	    IF (#i.ctrl.OFFVAL < #calc.speedmin) AND (#i.ctrl.ITLVAL > #calc.speedmax) THEN
	        #i.ctrl.OFFVAL := #calc.speedmin;
	    END_IF;
	    
	    //Network24: SPEED CONTROL: Determine if initialization routine is required
	    
	    #i.ctrl.init.req := (#i.ctrl.ITLVAL > #calc.speedmin) AND (#i.ctrl.init.dur < 0);
	    
	    //Network25: SPEED CONTROL: Determine the delay SP
	    
	    IF NOT #i.out.run AND #i.ctrl.init.req THEN
	        #i.ctrl.init.delay.in.spon := #i.ctrl.init.dur;
	    END_IF;
	    
	    IF NOT #i.out.run AND NOT #i.ctrl.init.req THEN
	        #i.ctrl.init.delay.in.spon := 0.0;
	    END_IF;
	    
	    IF #i.ctrl.mode OR NOT #ctrl_internal THEN
	        #i.ctrl.init.delay.in.spon := 0.0;
	    END_IF;
	    
	    //Network26: SPEED CONTROL: Delay for holding an init value
	    
	    "AFC_DelayONOFF"(cmd := #i.out.run,
	                     Pulse := #p100ms,
	                     Reset := NOT #i.out.run,
	                     on => #i.ctrl.init.delay.out.on,
	                     Data := #i.ctrl.init.delay);
	    
	    //Network27: SPEED CONTROL: Load output
	    
	    IF NOT #i.ctrl.mode THEN
	        
	        IF NOT #i.out.run THEN
	            
	            IF NOT #ctrl_internal THEN
	                
	                IF #i.ctrl.init.delay.out.on THEN
	                    #i.ctrl.OP := #i.scale.output;
	                END_IF;
	                
	                IF #i.ctrl.init.delay.out.on THEN
	                    #i.ctrl.OP := #i.ctrl.ITLVAL;
	                END_IF;
	                
	            END_IF;
	            
	        ELSIF NOT #ctrl_internal THEN
	            
	             #i.ctrl.OP := #i.ctrl.FUP;
	             
	        ELSE // 20240403: CH - Added "ELSE" for linear control
	             #i.ctrl.OP := #i.scale.output;
	            
	        END_IF;
	        
	    ELSIF #i.ctrl.mode THEN
	        
	         IF NOT #i.out.run AND NOT #i.ctrl.mode THEN
	            #i.ctrl.OP := #i.ctrl.OFFVAL;
	        END_IF;
	        
	    END_IF;
	    
	END_REGION
	
	REGION ARH  NW:28
	    
	    //Network28: ARH: Working hours counter
	    
	    IF #i.status.vfb AND #p1s THEN
	        #i.arh.seconds := #i.arh.seconds + 1;
	    END_IF;
	    
	    #i.arh.hour := #i.arh.seconds >= 3600;
	    
	    IF #i.arh.hour THEN
	        #i.arh.actual := #i.arh.actual + 1;
	        #i.arh.seconds := 0;
	    END_IF;
	    
	    IF #i.arh.resetarh THEN
	        #i.arh.actual := #i.arh.lastmaint := 0;
	    END_IF;
	    
	    #i.arh.difference := #i.arh.actual - #i.arh.lastmaint;
	    
	END_REGION
	
	REGION UNSCALE  NW:29-33
	    
	    //Network29: UNSCALE: Move input
	    
	    #i.unscale.in := #i.ctrl.OP;
	    
	    //Network30: UNSCALE: Cross-check unscaling setup
	    
	    #i.unscale.set := (#i.unscale.inhigh <> #i.unscale.inlow) AND (#i.unscale.outhigh <> #i.unscale.outlow);
	    
	    //Network31: UNSCALE: Determine sign of scaling slope and calculation operands (Hi - Low)
	    
	    IF #i.unscale.set THEN
	        #calc.inspan := #i.unscale.inhigh - #i.unscale.inlow;
	        #calc.outspan := #i.unscale.outhigh - #i.unscale.outlow;
	        #calc.x := #i.unscale.in;
	        IF #calc.inspan > 0 AND #calc.outspan > 0 THEN
	            #calc.sign := TRUE;
	            #calc.ymax := #i.unscale.outhigh;
	            #calc.ymin := #i.unscale.outlow;
	            #calc.xmax := #i.unscale.inhigh;
	            #calc.xmin := #i.unscale.inlow;
	        ELSIF #calc.inspan < 0 AND #calc.outspan < 0 THEN
	            #calc.sign := TRUE;
	            #calc.ymax := #i.unscale.outlow;
	            #calc.ymin := #i.unscale.outhigh;
	            #calc.xmax := #i.unscale.inlow;
	            #calc.xmin := #i.unscale.inhigh;
	        ELSIF #calc.inspan < 0 AND #calc.outspan > 0 THEN
	            #calc.sign := FALSE;
	            #calc.ymax := #i.unscale.outlow;
	            #calc.ymin := #i.unscale.outhigh;
	            #calc.xmax := #i.unscale.inhigh;
	            #calc.xmin := #i.unscale.inlow;
	        ELSE
	            #calc.sign := FALSE;
	            #calc.ymax := #i.unscale.outhigh;
	            #calc.ymin := #i.unscale.outlow;
	            #calc.xmax := #i.unscale.inlow;
	            #calc.xmin := #i.unscale.inhigh;
	        END_IF;
	        #calc.speedmin := #calc.xmin;
	        #calc.speedmax := #calc.xmax;
	    ELSE
	        #calc.inspan := #calc.outspan := #calc.xmax := #calc.xmin
	        := #calc.ymax := #calc.ymin := #calc.speedmin := #calc.speedmax := 0.0;
	    END_IF;
	    
	    //Network32: UNSCALE: Determine output
	    
	    IF #i.unscale.set AND #calc.sign THEN
	        
	        #calc.y := #calc.ymin + ((#calc.ymax - #calc.ymin) * (#calc.x - #calc.xmin) / (#calc.xmax - #calc.xmin));
	        
	        IF #calc.x <= #calc.xmin THEN
	            #calc.y := #calc.ymin;
	        END_IF;
	        
	        IF #calc.x >= #calc.xmax THEN
	            #calc.y := #calc.ymax;
	        END_IF;
	        
	    END_IF;
	    
	    IF #i.unscale.set AND NOT #calc.sign THEN
	        
	        #calc.y := #calc.ymin + ((#calc.ymax - #calc.ymin) * (#calc.xmax - #calc.x) / (#calc.xmax - #calc.xmin));
	        
	        IF #calc.x <= #calc.xmin THEN
	            #calc.y := #calc.ymax;
	        END_IF;
	        
	        IF #calc.x >= #calc.xmax THEN
	            #calc.y := #calc.ymin;
	        END_IF;
	        
	    END_IF;
	    
	    IF #i.unscale.set THEN
	        #i.unscale.output := #calc.y;
	    END_IF;
	    
	    IF NOT #i.unscale.set THEN
	        #i.unscale.output := 0.0;
	    END_IF;
	    
	    //Network33: UNSCALE: Convert to INT
	    
	    #i.out."ref" := REAL_TO_INT(#i.unscale.output);
	    
	END_REGION
	
	REGION UNSCALE  NW:34-35
	    
	    //Network34: ARH: Maintenance required
	    
	    #condSET := #i.arh.difference >= #i.arh.checkafter;
	    #condRESET := (#i.arh.completed AND #i.arh.maintenance) OR NOT #i.arh.enable;
	    
	    #i.arh.maintenance := (#i.arh.maintenance OR #condSET) AND NOT #condRESET;
	    
	    IF #i.arh.completed AND #i.arh.maintenance THEN
	        #i.arh.lastmaint := #i.arh.actual;
	    END_IF;
	    
	    
	    //Network35: STATUS: Maintenance required
	    
	    #i.status.maint := #i.arh.maintenance;
	    
	END_REGION
	
	REGION OUTPUT  NW:36
	    
	    //Network36: Move UDT outputs to FC outputs
	    
	    #run := #i.out.run;
	    #vfb := #i.status.vfb;
	    
	    #reference := #i.out."ref";
	    
	END_REGION
	
	REGION BUTTON  NW:37
	    
	    //Network37: EXTRA: Button treatment
	    
	    IF #i.ind.auto THEN
	        #i.cmd.auto := FALSE;
	    END_IF;
	    
	    IF #i.ind.man THEN
	        #i.cmd.man := FALSE;
	    END_IF;
	    
	    IF #i.ind.start OR #i.ind.auto OR NOT #i.status.ilstart THEN
	        #i.cmd.start := FALSE;
	    END_IF;
	    
	    IF #i.ind.stop OR #i.ind.auto THEN
	        #i.cmd.stop := FALSE;
	    END_IF;
	    
	    IF #i.faults.fpreset THEN
	        #i.faults.fpreset := FALSE;
	    END_IF;
	    
	    IF (#i.arh.seconds = 0) AND (#i.arh.actual = 0) THEN
	        #i.arh.resetarh := FALSE;
	    END_IF;
	    
	END_REGION
END_FUNCTION_BLOCK

FUNCTION_BLOCK "AFB_MotorPID_v3"
{ S7_Optimized_Access := 'TRUE' }
VERSION : 0.1
   VAR_INPUT 
      start { ExternalAccessible := 'False'; ExternalVisible := 'False'; ExternalWritable := 'False'} : Bool;   // "Logic" in order to start
      spsource { ExternalAccessible := 'False'; ExternalVisible := 'False'; ExternalWritable := 'False'} : Bool;   // 0=internal setpoint, 1=external setpoint
      followup { ExternalAccessible := 'False'; ExternalVisible := 'False'; ExternalWritable := 'False'} : Bool;   // 0=motor control from PID, 1=motor setpoint directly from program
      pidrun { ExternalAccessible := 'False'; ExternalVisible := 'False'; ExternalWritable := 'False'} : Bool;   // 0=controller not ready, controller is running
      "fb" { ExternalAccessible := 'False'; ExternalVisible := 'False'; ExternalWritable := 'False'} : Bool;   // Motor's running feedback (1=run, 0=stop)
      mcb { ExternalAccessible := 'False'; ExternalVisible := 'False'; ExternalWritable := 'False'} : Bool;   // Motor circuit breaker (1=ok, 0=fault)
      ctrl { ExternalAccessible := 'False'; ExternalVisible := 'False'; ExternalWritable := 'False'} : Bool;   // Control of motor (1=PLC, 0=Local)
      vfdnotrip { ExternalAccessible := 'False'; ExternalVisible := 'False'; ExternalWritable := 'False'} : Bool;   // VFD health condition (1=ok, 0=fault)
      block { ExternalAccessible := 'False'; ExternalVisible := 'False'; ExternalWritable := 'False'} : Bool;   // Condition that blocks motor operation
      generalackn { ExternalAccessible := 'False'; ExternalVisible := 'False'; ExternalWritable := 'False'} : Bool;   // General acknowledgement
      reset { ExternalAccessible := 'False'; ExternalVisible := 'False'; ExternalWritable := 'False'} : Bool;   // Option that resets the faults
      mute { ExternalAccessible := 'False'; ExternalVisible := 'False'; ExternalWritable := 'False'} : Bool;   // Mute siren
      autoset { ExternalAccessible := 'False'; ExternalVisible := 'False'; ExternalWritable := 'False'} : Bool;   // Option that sets the motor to auto mode (Used for mass auto set)
      manualset { ExternalAccessible := 'False'; ExternalVisible := 'False'; ExternalWritable := 'False'} : Bool;   // Option that sets the motor to manual mode (Used for mass manual set)
      p1s { ExternalAccessible := 'False'; ExternalVisible := 'False'; ExternalWritable := 'False'} : Bool;   // Pulse that is generated every 1 s (Count up)
      p100ms { ExternalAccessible := 'False'; ExternalVisible := 'False'; ExternalWritable := 'False'} : Bool;   // Pulse that is generated every 100 ms (Count up)
      blink { ExternalAccessible := 'False'; ExternalVisible := 'False'; ExternalWritable := 'False'} : Bool;   // Blink that is used for the graphics (Frequency of CPU)
      PV { ExternalAccessible := 'False'; ExternalVisible := 'False'; ExternalWritable := 'False'} : Real;   // Peripheral value reference to the controller
      PV_unit { ExternalAccessible := 'False'; ExternalVisible := 'False'; ExternalWritable := 'False'} : WString;   // Peripheral value unit
      EXT_SP { ExternalAccessible := 'False'; ExternalVisible := 'False'; ExternalWritable := 'False'} : Real;   // External setpoint
      FUP { ExternalAccessible := 'False'; ExternalVisible := 'False'; ExternalWritable := 'False'} : Real;   // Follow up value
      Out_unit { ExternalAccessible := 'False'; ExternalVisible := 'False'; ExternalWritable := 'False'} : WString;   // Output unit (If nothing is entered then it is from the HMI)
   END_VAR

   VAR_OUTPUT 
      run { ExternalAccessible := 'False'; ExternalVisible := 'False'; ExternalWritable := 'False'} : Bool;   // Command to start motor
      vfb { ExternalAccessible := 'False'; ExternalVisible := 'False'; ExternalWritable := 'False'} : Bool;   // Virtual feedback (used everywhere instead of digital fb)
      reference { ExternalAccessible := 'False'; ExternalVisible := 'False'; ExternalWritable := 'False'} : Int;   // Reference to analog output card
   END_VAR

   VAR_IN_OUT 
      faults : "UDT_MTRFAULTS";   // External data (Primary alarm data - alarm & plc ackn)
   END_VAR

   VAR RETAIN
      i : "UDT_MOTOR";   // Data type containing the motor's data
   END_VAR
   VAR 
      cont { ExternalAccessible := 'False'; ExternalVisible := 'False'; ExternalWritable := 'False'} : Struct   // Controller
         COM_RST { ExternalAccessible := 'False'; ExternalVisible := 'False'; ExternalWritable := 'False'} : Bool;   // Restart command
         MAN_ON { ExternalAccessible := 'False'; ExternalVisible := 'False'; ExternalWritable := 'False'} : Bool;   // Manual control
         SP_INT { ExternalAccessible := 'False'; ExternalVisible := 'False'; ExternalWritable := 'False'} : Real;   // Setpoint internal
         PV_IN { ExternalAccessible := 'False'; ExternalVisible := 'False'; ExternalWritable := 'False'} : Real;   // Peripheral value
         GAIN { ExternalAccessible := 'False'; ExternalVisible := 'False'; ExternalWritable := 'False'} : Real;   // Proportional gain loaded according to the action (signed)
         TI { ExternalAccessible := 'False'; ExternalVisible := 'False'; ExternalWritable := 'False'} : Time;   // Integral time
         TD { ExternalAccessible := 'False'; ExternalVisible := 'False'; ExternalWritable := 'False'} : Time;   // Derivative time
         LMN_HLM { ExternalAccessible := 'False'; ExternalVisible := 'False'; ExternalWritable := 'False'} : Real;   // Controller's higher LMN value (%)
         LMN_LLM { ExternalAccessible := 'False'; ExternalVisible := 'False'; ExternalWritable := 'False'} : Real;   // Controller's lower LMN value (%)
         LMN_FAC { ExternalAccessible := 'False'; ExternalVisible := 'False'; ExternalWritable := 'False'} : Real;   // LMN factor
         LMN_OFF { ExternalAccessible := 'False'; ExternalVisible := 'False'; ExternalWritable := 'False'} : Real;   // LMN offset
         I_ITLVAL { ExternalAccessible := 'False'; ExternalVisible := 'False'; ExternalWritable := 'False'} : Real;   // Controller's integral initialization value (%)
         LMN { ExternalAccessible := 'False'; ExternalVisible := 'False'; ExternalWritable := 'False'} : Real;   // Controller's manipulated value
      END_STRUCT;
      calc { ExternalAccessible := 'False'; ExternalVisible := 'False'; ExternalWritable := 'False'} : Struct   // Calculations for scaling process
         inspan { ExternalAccessible := 'False'; ExternalVisible := 'False'; ExternalWritable := 'False'} : Real;   // Scaling span
         outspan { ExternalAccessible := 'False'; ExternalVisible := 'False'; ExternalWritable := 'False'} : Real;   // Channel span
         xmax { ExternalAccessible := 'False'; ExternalVisible := 'False'; ExternalWritable := 'False'} : Real;   // Channel maximum value
         xmin { ExternalAccessible := 'False'; ExternalVisible := 'False'; ExternalWritable := 'False'} : Real;   // Channel minimum value
         ymax { ExternalAccessible := 'False'; ExternalVisible := 'False'; ExternalWritable := 'False'} : Real;   // Output maximum value
         ymin { ExternalAccessible := 'False'; ExternalVisible := 'False'; ExternalWritable := 'False'} : Real;   // Output minimum value
         x { ExternalAccessible := 'False'; ExternalVisible := 'False'; ExternalWritable := 'False'} : Real;   // Active x value (channel)
         y { ExternalAccessible := 'False'; ExternalVisible := 'False'; ExternalWritable := 'False'} : Real;   // Active y value (output)
         sign { ExternalAccessible := 'False'; ExternalVisible := 'False'; ExternalWritable := 'False'} : Bool;   // Linear scaling slope sign
      END_STRUCT;
   END_VAR

   VAR_TEMP 
      condSET : Bool;
      condRESET : Bool;
   END_VAR


BEGIN
	REGION GEN  NW:2
	    
	    //Network2: GEN: Move FB inputs to UDT inputs
	    
	    #i.pid.spsource := #spsource;
	    #i.pid.followup := #followup;
	    #i.pid.pidrun := #pidrun;
	    #i.pid.PV := #PV;
	    #i.pid.EXT_SP := #EXT_SP;
	    #i.pid.FUP := #FUP;
	    #i.pid.pvunit := #PV_unit;
	    
	    IF #PV_unit <> WSTRING#'' THEN
	        #i.pid.pvunit := #PV_unit;
	    END_IF;
	    
	    IF #Out_unit <> WSTRING#'' THEN
	        #i.pid.outunit := #Out_unit;
	    END_IF;
	    
	END_REGION
	
	REGION STATUS  NW:3-4
	    
	    //Network3: STATUS: Virtual feedback
	    
	    #i.status.vfb := (#fb AND NOT #i.sim.fb) OR (#i.out.run AND #i.sim.fb);
	    
	    //Network4: STATUS: Virtual control
	    
	    #i.status.vctrl := #i.sim.ctrl OR (#ctrl AND NOT #i.sim.ctrl);
	    
	END_REGION
	
	REGION FAULT  NW:5-10
	    
	    //Network5: FAULT: Fail to run
	    
	    "AFC_AlarmAckn"(trigger := NOT #i.status.vfb AND #i.out.run AND #i.status.vctrl,
	                    release := NOT #i.sim.fb,
	                    ctrlpoint := FALSE,
	                    enackn := TRUE,
	                    ensiren := TRUE,
	                    p100ms := #p100ms,
	                    generalackn := #generalackn OR #i.faults.fpreset,
	                    reset := #reset OR #i.faults.fpreset,
	                    mute := #mute,
	                    delay := 0.0,
	                    plcackn => #faults.ctrl.plcackn_ftr,
	                    alarm => #faults.ctrl.alarm_ftr,
	                    siren => #faults.status.siren_ftr,
	                    hmiackn := #faults.status.hmiackn_ftr,
	                    Data := #i.faults.ftr);
	    
	    //Network6: FAULT: Fail to stop
	    
	    "AFC_AlarmAckn"(trigger := #i.status.vfb AND NOT #i.out.run AND #i.status.vctrl,
	                    release := NOT #i.sim.fb,
	                    ctrlpoint := FALSE,
	                    enackn := TRUE,
	                    ensiren := TRUE,
	                    p100ms := #p100ms,
	                    generalackn := #generalackn OR #i.faults.fpreset,
	                    reset := #reset OR #i.faults.fpreset,
	                    mute := #mute,
	                    delay := 0.0,
	                    plcackn => #faults.ctrl.plcackn_fts,
	                    alarm => #faults.ctrl.alarm_fts,
	                    siren => #faults.status.siren_fts,
	                    hmiackn := #faults.status.hmiackn_fts,
	                    Data := #i.faults.fts);
	    
	    //Network7: FAULT: Monor circuit breaker
	    
	    "AFC_AlarmAckn"(trigger := NOT #mcb,
	                    release := NOT #i.sim.fb,
	                    ctrlpoint := FALSE,
	                    enackn := TRUE,
	                    ensiren := TRUE,
	                    p100ms := #p100ms,
	                    generalackn := #generalackn OR #i.faults.fpreset,
	                    reset := #reset OR #i.faults.fpreset,
	                    mute := #mute,
	                    delay := 0.0,
	                    plcackn => #faults.ctrl.plcackn_mcb,
	                    alarm => #faults.ctrl.alarm_mcb,
	                    siren => #faults.status.siren_mcb,
	                    hmiackn := #faults.status.hmiackn_mcb,
	                    Data := #i.faults.mcb);
	    
	    //Network8: FAULT: Control
	    
	    "AFC_AlarmAckn"(trigger := NOT #i.status.vctrl AND #i.out.run,
	                    release := NOT #i.sim.ctrl,
	                    ctrlpoint := FALSE,
	                    enackn := TRUE,
	                    ensiren := TRUE,
	                    p100ms := #p100ms,
	                    generalackn := #generalackn OR #i.faults.fpreset,
	                    reset := #reset OR #i.faults.fpreset,
	                    mute := #mute,
	                    delay := 0.0,
	                    plcackn => #faults.ctrl.plcackn_ctrl,
	                    alarm => #faults.ctrl.alarm_ctrl,
	                    siren => #faults.status.siren_ctrl,
	                    hmiackn := #faults.status.hmiackn_ctrl,
	                    Data := #i.faults.ctrl);
	    
	    //Network9: FAULT: Variable frequency drive
	    
	    "AFC_AlarmAckn"(trigger := NOT #vfdnotrip,
	                    release := TRUE,
	                    ctrlpoint := FALSE,
	                    enackn := TRUE,
	                    ensiren := TRUE,
	                    p100ms := #p100ms,
	                    generalackn := #generalackn OR #i.faults.fpreset,
	                    reset := #reset OR #i.faults.fpreset,
	                    mute := #mute,
	                    delay := 0.0,
	                    plcackn => #faults.ctrl.plcackn_vfd,
	                    alarm => #faults.ctrl.alarm_vfd,
	                    siren => #faults.status.siren_vfd,
	                    hmiackn := #faults.status.hmiackn_vfd,
	                    Data := #i.faults.vfd);
	    
	    //Network10: FAULT: Interlock violation
	    
	    "AFC_AlarmAckn"(trigger := #start AND #block,
	                    release := #i.status.ilstart,
	                    ctrlpoint := FALSE,
	                    enackn := TRUE,
	                    ensiren := TRUE,
	                    p100ms := #p100ms,
	                    generalackn := #generalackn OR #i.faults.fpreset,
	                    reset := #reset OR #i.faults.fpreset,
	                    mute := #mute,
	                    delay := 0.0,
	                    plcackn => #faults.ctrl.plcackn_il,
	                    alarm => #faults.ctrl.alarm_il,
	                    siren => #faults.status.siren_il,
	                    hmiackn := #faults.status.hmiackn_il,
	                    Data := #i.faults.il);
	    
	END_REGION
	
	REGION STATUS  NW:11-12
	    
	    //Network11: STATUS: General Fault
	    
	    #i.status.fault := #i.faults.ftr.status.alarm OR #i.faults.fts.status.alarm OR #i.faults.mcb.status.alarm OR #i.faults.ctrl.status.alarm OR #i.faults.vfd.status.alarm OR #i.faults.il.status.alarm;
	    
	    //Network12: STATUS: Start interlock
	    
	    #i.status.ilstart := NOT (#block OR #i.status.fault) AND #i.status.vctrl AND #i.unscale.set;
	    
	END_REGION
	
	REGION CONTROL  NW:13-15
	    
	    //Network13: CONTROL: Manual Set
	    
	    #condSET := #i.cmd.man OR #manualset;
	    #condRESET := #i.cmd.auto OR #autoset;
	    
	    #i.ind.man := (#i.ind.man OR #condSET) AND NOT #condRESET;
	    
	    //Network14: CONTROL: Auto Set
	    
	    #i.ind.auto := NOT #i.ind.man;
	    
	    //Network15: CONTROL: Manual Run
	    
	    #condSET := #i.cmd.start AND #i.ind.man;
	    #condRESET := #i.cmd.stop OR (NOT #i.ind.man) AND (NOT #i.status.ilstart);
	    
	    #i.out.manrun := (#i.out.manrun OR #condSET) AND NOT #condRESET;
	    
	END_REGION
	
	REGION STATUS  NW:16-17
	    
	    //Network16: STATUS: Motor's icon
	    
	    #i.status.icon := 0;
	    
	    IF #i.status.vfb AND NOT #i.status.fault AND #i.status.vctrl
	    THEN
	        #i.status.icon := 1;
	    ELSIF #fb AND NOT #i.status.fault AND NOT #i.status.vctrl
	    THEN
	        #i.status.icon := 2;
	    ELSIF #i.status.fault AND #blink
	    THEN
	        #i.status.icon := 3;
	    END_IF;
	    
	    //Network17: STATUS:Start/Stop Buttons
	    
	    #i.ind.start := #i.out.manrun AND #i.ind.man;
	    #i.ind.stop := NOT #i.out.manrun AND #i.ind.man;
	    
	END_REGION
	
	REGION OUTPUT  NW:18
	    
	    //Network18: OUTPUT: Start motor
	    
	    #condSET := #i.status.ilstart AND (#i.out.manrun OR (#start AND #i.ind.auto));
	    #condRESET := NOT #i.status.ilstart;
	    
	    "AFC_DelayONOFF"(cmd := #condSET,
	                     Pulse := #p100ms,
	                     Reset := #condRESET,
	                     on => #i.out.run,
	                     Data := #i.delay);
	    
	END_REGION
	
	REGION CONTROLLER  NW:19
	    
	    //Network19: CONTROLLER: Load from PID block
	    
	    #i.pid.LMN := #cont.LMN;
	    
	END_REGION
	
	REGION PID  NW:20-27
	    
	    //Network20: PID: Manage controller's limits
	    
	    IF #i.pid.H <= #i.pid.L THEN
	        #i.pid.H := #i.pid.L := #calc.xmin;
	    END_IF;
	    
	    IF #i.pid.H > #calc.xmax THEN
	        #i.pid.H := #calc.xmax;
	    END_IF;
	    
	    IF #i.pid.L < #calc.xmin THEN
	        #i.pid.L := #calc.xmin;
	    END_IF;
	    
	    IF (#i.pid.ITLVAL < #i.pid.L) AND (#i.pid.ITLVAL > #i.pid.H) THEN
	        #i.pid.ITLVAL := #calc.xmin;
	    END_IF;
	    
	    IF (#i.pid.OFFVAL < #i.pid.L) AND (#i.pid.ITLVAL > #i.pid.H) THEN
	        #i.pid.OFFVAL := #calc.xmin;
	    END_IF;
	    
	    
	    //Network21: PID: Load SP
	    
	    IF #i.pid.spsource THEN
	        #i.pid.SP := #i.pid.EXT_SP;
	    END_IF;
	    
	    
	    //Network22: PID: Determine if initialization routine is required
	    
	    #i.pid.init.req := (#i.pid.ITLVAL > #i.pid.L) AND (#i.pid.init.dur > 0.0);
	    
	    //Network23: PID: Determine the delay SP
	    
	    IF NOT #i.out.run AND #i.pid.init.req THEN
	        #i.pid.init.delay.in.spon := #i.pid.init.dur;
	    END_IF;
	    
	    IF NOT #i.out.run AND NOT #i.pid.init.req THEN
	        #i.pid.init.delay.in.spon := 0.0;
	    END_IF;
	    
	    IF #i.pid.mode = #i.pid.followup THEN
	        #i.pid.init.delay.in.spon := 0.0;
	    END_IF;
	    
	    
	    //Network24: PID: Delay for holding an init value
	    
	    "AFC_DelayONOFF"(cmd := #i.out.run,
	                     Pulse := #p100ms,
	                     Reset := NOT #i.out.run,
	                     on => #i.pid.init.delay.out.on,
	                     Data := #i.pid.init.delay);
	    
	    //Network25: PID: Reset the controller
	    
	    #i.pid.cmdrst := NOT #i.pid.init.delay.out.on OR #i.pid.mode OR #i.pid.followup;
	    
	    //Network26: PID: Load output
	    
	    IF NOT #i.pid.mode THEN
	        
	        IF #i.out.run THEN
	            
	            IF NOT #i.pid.followup THEN
	                
	                IF #i.pid.pidrun THEN
	                    #i.pid.OP := #i.pid.LMN;
	                END_IF;
	                
	                IF #i.pid.cmdrst THEN
	                    #i.pid.OP := #i.pid.ITLVAL;
	                END_IF;
	                
	            ELSIF #i.pid.followup THEN
	                
	                #i.pid.OP := #i.pid.FUP;
	                
	            END_IF;
	            
	        END_IF;
	        
	        IF NOT #i.out.run THEN
	            #i.pid.OP := #i.pid.OFFVAL;
	        END_IF;
	        ;
	        
	    END_IF;
	    
	    //Network27: PID: Limit output
	    
	    IF #i.pid.OP < #calc.xmin THEN
	        #i.pid.OP := #calc.xmin;
	    END_IF;
	    
	    IF #i.pid.OP > #calc.xmax THEN
	        #i.pid.OP := #calc.xmax;
	    END_IF;
	    
	END_REGION
	
	REGION UNSCALE  NW:28-32
	    
	    //Network28: UNSCALE: Move input
	    
	    #i.unscale.in := #i.pid.OP;
	    
	    //Network29: UNSCALE: Cross-check unscaling setup
	    
	    #i.unscale.set := (#i.unscale.inhigh <> #i.unscale.inlow) AND (#i.unscale.outhigh <> #i.unscale.outlow);
	    
	    //Network30: UNSCALE: Determine sign of scaling slope and calculation operands (Hi - Low)
	    
	    IF #i.unscale.set THEN
	        #calc.inspan := #i.unscale.inhigh - #i.unscale.inlow;
	        #calc.outspan := #i.unscale.outhigh - #i.unscale.outlow;
	        #calc.x := #i.unscale.in;
	        IF #calc.inspan > 0 AND #calc.outspan > 0 THEN
	            #calc.sign := TRUE;
	            #calc.ymax := #i.unscale.outhigh;
	            #calc.ymin := #i.unscale.outlow;
	            #calc.xmax := #i.unscale.inhigh;
	            #calc.xmin := #i.unscale.inlow;
	        ELSIF #calc.inspan < 0 AND #calc.outspan < 0 THEN
	            #calc.sign := TRUE;
	            #calc.ymax := #i.unscale.outlow;
	            #calc.ymin := #i.unscale.outhigh;
	            #calc.xmax := #i.unscale.inlow;
	            #calc.xmin := #i.unscale.inhigh;
	        ELSIF #calc.inspan < 0 AND #calc.outspan > 0 THEN
	            #calc.sign := FALSE;
	            #calc.ymax := #i.unscale.outlow;
	            #calc.ymin := #i.unscale.outhigh;
	            #calc.xmax := #i.unscale.inhigh;
	            #calc.xmin := #i.unscale.inlow;
	        ELSE
	            #calc.sign := FALSE;
	            #calc.ymax := #i.unscale.outhigh;
	            #calc.ymin := #i.unscale.outlow;
	            #calc.xmax := #i.unscale.inlow;
	            #calc.xmin := #i.unscale.inhigh;
	        END_IF;
	    ELSE
	        #calc.inspan := #calc.outspan := #calc.xmax := #calc.xmin := #calc.ymax := #calc.ymin := 0;
	    END_IF;
	    
	    //Network31: UNSCALE: Determine output
	    
	    IF #i.unscale.set AND #calc.sign THEN
	        
	        #calc.y := #calc.ymin + ((#calc.ymax - #calc.ymin) * (#calc.x - #calc.xmin) / (#calc.xmax - #calc.xmin));
	        
	        IF #calc.x <= #calc.xmin THEN
	            #calc.y := #calc.ymin;
	        END_IF;
	        
	        IF #calc.x >= #calc.xmax THEN
	            #calc.y := #calc.ymax;
	        END_IF;
	        
	    END_IF;
	    
	    IF #i.unscale.set AND NOT #calc.sign THEN
	        
	        #calc.y := #calc.ymin + ((#calc.ymax - #calc.ymin) * (#calc.xmax - #calc.x) / (#calc.xmax - #calc.xmin));
	        
	        IF #calc.x <= #calc.xmin THEN
	            #calc.y := #calc.ymax;
	        END_IF;
	        
	        IF #calc.x >= #calc.xmax THEN
	            #calc.y := #calc.ymin;
	        END_IF;
	        
	    END_IF;
	    
	    IF #i.unscale.set THEN
	        #i.unscale.output := #calc.y;
	    END_IF;
	    
	    IF NOT #i.unscale.set THEN
	        #i.unscale.output := 0.0;
	    END_IF;
	    
	    //Network32: UNSCALE: Convert to INT
	    
	    #i.out."ref" := REAL_TO_INT(#i.unscale.output);
	    
	END_REGION
	
	REGION CONTROLLER  NW:33
	    
	    //Network33: CONTROLLER: Load to PID block
	    
	    #cont.COM_RST := #i.pid.cmdrst;
	    
	    #cont.MAN_ON := #i.pid.mode;
	    
	    #cont.SP_INT := #i.pid.SP;
	    
	    #cont.PV_IN := #i.pid.PV;
	    
	    IF #i.pid.action THEN
	        #cont.GAIN := ABS_REAL(#i.pid.P);
	    ELSE
	        #cont.GAIN := 0.0 - ABS_REAL(#i.pid.P);
	    END_IF;
	    
	    #cont.TI := DINT_TO_TIME(#i.pid.I);
	    
	    #cont.TD := DINT_TO_TIME(#i.pid.D);
	    
	    #cont.LMN_HLM := ((#i.pid.H - #calc.xmin) / (#calc.xmax - #calc.xmin)) * 100.0;
	    
	    #cont.LMN_LLM := ((#i.pid.L - #calc.xmin) / (#calc.xmax - #calc.xmin)) * 100.0;
	    
	    #cont.LMN_FAC := (#calc.xmax - #calc.xmin) / 100.0;
	    
	    #cont.LMN_OFF := #calc.xmin;
	    
	    #cont.I_ITLVAL := ((#i.pid.OP - #calc.xmin) / (#calc.xmax - #calc.xmin)) * 100.0;
	    
	END_REGION
	
	
	REGION MNT  NW:34-36
	    
	    //Network34: ARH: Working hours counter
	    
	    IF #i.status.vfb AND #p1s THEN
	        #i.arh.seconds := #i.arh.seconds + 1;
	    END_IF;
	    
	    #i.arh.hour := (#i.arh.seconds >= 3600);
	    
	    IF #i.arh.hour THEN
	        #i.arh.actual := #i.arh.actual + 1;
	        #i.arh.seconds := 0;
	    END_IF;
	    
	    IF #i.arh.resetarh THEN
	        #i.arh.actual := #i.arh.lastmaint := 0;
	    END_IF;
	    
	    #i.arh.difference := #i.arh.actual - #i.arh.lastmaint;
	    
	    //Network35: ARH: Maintenance required
	    
	    #condSET := #i.arh.difference >= #i.arh.checkafter;
	    #condRESET := (#i.arh.completed AND #i.arh.maintenance) OR NOT #i.arh.enable;
	    
	    #i.arh.maintenance := (#i.arh.maintenance OR #condSET) AND NOT #condRESET;
	    
	    IF #i.arh.completed AND #i.arh.maintenance THEN
	        #i.arh.lastmaint := #i.arh.actual;
	    END_IF;
	    
	    //Network36: STATUS: Maintenance required
	    
	    #i.status.maint := #i.arh.maintenance;
	    
	END_REGION
	
	REGION OUTPUT  NW:37
	    
	    //Network37: Move UDT outputs to FC outputs
	    
	    #run := #i.out.run;
	    #vfb := #i.status.vfb;
	    
	    #reference := #i.out."ref";
	    
	END_REGION
	
	REGION BUTTON  NW:38
	    
	    //Network38: EXTRA: Button treatment
	    
	    IF #i.ind.auto THEN
	        #i.cmd.auto := FALSE;
	    END_IF;
	    
	    IF #i.ind.man THEN
	        #i.cmd.man := FALSE;
	    END_IF;
	    
	    IF #i.ind.start OR #i.ind.auto OR NOT #i.status.ilstart THEN
	        #i.cmd.start := FALSE;
	    END_IF;
	    
	    IF #i.ind.stop OR #i.ind.auto THEN
	        #i.cmd.stop := FALSE;
	    END_IF;
	    
	    IF #i.faults.fpreset THEN
	        #i.faults.fpreset := FALSE;
	    END_IF;
	    
	    IF (#i.arh.seconds = 0) AND (#i.arh.actual = 0) THEN
	        #i.arh.resetarh := FALSE;
	    END_IF;
	    
	END_REGION
END_FUNCTION_BLOCK

FUNCTION_BLOCK "AFB_Valve_v3"
{ S7_Optimized_Access := 'TRUE' }
VERSION : 0.1
   VAR_INPUT 
      actmain { ExternalAccessible := 'False'; ExternalVisible := 'False'; ExternalWritable := 'False'} : Bool;   // Command to open the valve's main route
      actupper { ExternalAccessible := 'False'; ExternalVisible := 'False'; ExternalWritable := 'False'} : Bool;   // Command to open the valve's upper s/l route
      actlower { ExternalAccessible := 'False'; ExternalVisible := 'False'; ExternalWritable := 'False'} : Bool;   // Command to open the valve's lower s/l route
      fbmain { ExternalAccessible := 'False'; ExternalVisible := 'False'; ExternalWritable := 'False'} : Bool;   // Feedback that indicates that the valve's main route is activated
      fbupper { ExternalAccessible := 'False'; ExternalVisible := 'False'; ExternalWritable := 'False'} : Bool;   // Feedback that indicates that the valve's upper s/l route is activated
      fblower { ExternalAccessible := 'False'; ExternalVisible := 'False'; ExternalWritable := 'False'} : Bool;   // Feedback that indicates that the valve's lower s/l route is activated
      fbdeact { ExternalAccessible := 'False'; ExternalVisible := 'False'; ExternalWritable := 'False'} : Bool;   // Feedback that indicates that the valve is deactivated
      blockmain { ExternalAccessible := 'False'; ExternalVisible := 'False'; ExternalWritable := 'False'} : Bool;   // Interlock that blocks valve's main activation
      blockupper { ExternalAccessible := 'False'; ExternalVisible := 'False'; ExternalWritable := 'False'} : Bool;   // Interlock that blocks valve's upper s/l activation
      blocklower { ExternalAccessible := 'False'; ExternalVisible := 'False'; ExternalWritable := 'False'} : Bool;   // Interlock that blocks valve's lower s/l activation
      generalackn { ExternalAccessible := 'False'; ExternalVisible := 'False'; ExternalWritable := 'False'} : Bool;   // General acknowledgement
      reset { ExternalAccessible := 'False'; ExternalVisible := 'False'; ExternalWritable := 'False'} : Bool;   // Option that resets the faults
      mute { ExternalAccessible := 'False'; ExternalVisible := 'False'; ExternalWritable := 'False'} : Bool;   // Mute siren
      autoset { ExternalAccessible := 'False'; ExternalVisible := 'False'; ExternalWritable := 'False'} : Bool;   // Extra option that sets the valve in auto mode (ex. group set)
      manualset { ExternalAccessible := 'False'; ExternalVisible := 'False'; ExternalWritable := 'False'} : Bool;   // Extra option that sets the valve in manual mode (ex. group set)
      p1s { ExternalAccessible := 'False'; ExternalVisible := 'False'; ExternalWritable := 'False'} : Bool;   // Pulse that is generated every 1 s
      p100ms { ExternalAccessible := 'False'; ExternalVisible := 'False'; ExternalWritable := 'False'} : Bool;   // Pulse that is generated every 100 ms
      blink { ExternalAccessible := 'False'; ExternalVisible := 'False'; ExternalWritable := 'False'} : Bool;   // Blink used for the graphics
      "type" { ExternalAccessible := 'False'; ExternalVisible := 'False'; ExternalWritable := 'False'} : Int;   // 0=1Q, 1= 3Q
   END_VAR

   VAR_OUTPUT 
      main { ExternalAccessible := 'False'; ExternalVisible := 'False'; ExternalWritable := 'False'} : Bool;   // Activate main route
      upper { ExternalAccessible := 'False'; ExternalVisible := 'False'; ExternalWritable := 'False'} : Bool;   // Activate upper s/l route
      lower { ExternalAccessible := 'False'; ExternalVisible := 'False'; ExternalWritable := 'False'} : Bool;   // Activate lower s/l route
      vfbmain { ExternalAccessible := 'False'; ExternalVisible := 'False'; ExternalWritable := 'False'} : Bool;   // Virtual feedback - Activated main route
      vfbupper { ExternalAccessible := 'False'; ExternalVisible := 'False'; ExternalWritable := 'False'} : Bool;   // Virtual feedback - Activated upper s/l route
      vfblower { ExternalAccessible := 'False'; ExternalVisible := 'False'; ExternalWritable := 'False'} : Bool;   // Virtual feedback - Activated lower s/l route
      vfbdeact { ExternalAccessible := 'False'; ExternalVisible := 'False'; ExternalWritable := 'False'} : Bool;   // Virtual feedback - Deactivated
   END_VAR

   VAR_IN_OUT 
      faults : "UDT_VALVEFAULTS";   // External data (Primary alarm data - alarm & plc ackn)
   END_VAR

   VAR RETAIN
      i : "UDT_VALVE";
   END_VAR

   VAR_TEMP 
      condSET : Bool;
      condRESET : Bool;
   END_VAR


BEGIN
	REGION FEEDBACK  NW:2-5
	    
	    //Network2: FEEDBACK: Generate virtual (processed) feedback (main route)
	    
	    #i.status.vfbmain := (#fbmain AND NOT #i.sim.main) OR (#i.out.actmain AND #i.sim.main);
	    
	    //Network3: FEEDBACK: Generate virtual (processed) feedback (upper s/l route)
	    
	    #i.status.vfbupper := (#fbupper AND NOT #i.sim.upper) OR (#i.out.actupper AND #i.sim.upper);
	    
	    //Network4: FEEDBACK: Generate virtual (processed) feedback (lower s/l route)
	    
	    #i.status.vfblower := (#fblower AND NOT #i.sim.lower) OR (#i.out.actlower AND #i.sim.lower);
	    
	    //Network5: FEEDBACK: Generate virtual (processed) feedback (deactivated)
	    
	    #i.status.vfbdeact := (#fbdeact AND NOT #i.sim.deact) OR (NOT #i.out.actmain AND NOT #i.out.actlower AND NOT #i.out.actupper AND NOT #i.sim.deact);
	    
	END_REGION
	
	REGION MANUAL CONTROL  NW:6-10
	    
	    //Network6: MANUAL CONTROL: Manual set
	    
	    #condSET := #i.cmd.man OR #manualset;
	    #condRESET := #i.cmd.auto OR #autoset;
	    
	    #i.ind.man := (#i.ind.man OR #condSET) AND NOT #condRESET;
	    
	    //Network7: MANUAL CONTROL: Auto set
	    
	    #i.ind.auto := NOT #i.ind.man;
	    
	    //Network8: MANUAL CONTROL: Activate manually main route
	    
	    #condSET := NOT (#i.man.upper OR #i.man.lower OR #i.cmd.upper OR #i.cmd.lower) AND (#i.ind.man AND #i.cmd.main);
	    #condRESET := #i.cmd.deact OR NOT (#i.status.ilactmain AND #i.ind.man);
	    
	    #i.man.main := (#i.man.main OR #condSET) AND NOT #condRESET;
	    
	    //Network9: MANUAL CONTROL: Activate manually upper s/l route
	    
	    #condSET := NOT (#i.man.main OR #i.man.lower OR #i.cmd.main OR #i.cmd.lower) AND (#i.ind.man AND #i.cmd.upper);
	    #condRESET := #i.cmd.deact OR (#type <> 1) OR NOT (#i.status.ilactupper AND #i.ind.man);
	    
	    #i.man.upper := (#i.man.upper OR #condSET) AND NOT #condRESET;
	    
	    //Network10: MANUAL CONTROL: Activate manually lower s/l route
	    
	    #condSET := NOT (#i.man.upper OR #i.man.main OR #i.cmd.upper OR #i.cmd.main) AND (#i.ind.man AND #i.cmd.lower);
	    #condRESET := #i.cmd.deact OR (#type <> 1) OR NOT (#i.status.ilactlower AND #i.ind.man);
	    
	    #i.man.lower := (#i.man.lower OR #condSET) AND NOT #condRESET;
	    
	END_REGION
	
	REGION FAULT  NW:11-15
	    
	    //Network11: FAULT: Fail to activate main route
	    
	    "AFC_AlarmAckn"(trigger := (NOT #i.status.vfbmain AND #i.out.actmain) OR (#i.status.vfbdeact AND #i.out.actmain),
	                    release := NOT #i.sim.main,
	                    ctrlpoint := FALSE,
	                    enackn := TRUE,
	                    ensiren := TRUE,
	                    p100ms := #p100ms,
	                    generalackn := #generalackn OR #i.faults.fpreset,
	                    reset := #reset OR #i.faults.fpreset,
	                    mute := #mute,
	                    delay := 0.0,
	                    plcackn => #faults.ctrl.plcackn_ftamain,
	                    alarm => #faults.ctrl.alarm_ftamain,
	                    siren => #faults.status.siren_ftamain,
	                    hmiackn := #faults.status.hmiackn_ftamain,
	                    Data := #i.faults.ftamain);
	    
	    //Network12: FAULT: Fail to activate upper route
	    
	    "AFC_AlarmAckn"(trigger := NOT #i.status.vfbupper AND #i.out.actupper,
	                    release := NOT #i.sim.upper AND #type = 1,
	                    ctrlpoint := FALSE,
	                    enackn := TRUE,
	                    ensiren := TRUE,
	                    p100ms := #p100ms,
	                    generalackn := #generalackn OR #i.faults.fpreset,
	                    reset := #reset OR #i.faults.fpreset,
	                    mute := #mute,
	                    delay := 0.0,
	                    plcackn => #faults.ctrl.plcackn_ftaupper,
	                    alarm => #faults.ctrl.alarm_ftaupper,
	                    siren => #faults.status.siren_ftaupper,
	                    hmiackn := #faults.status.hmiackn_ftaupper,
	                    Data := #i.faults.ftaupper);
	    
	    //Network13: FAULT: Fail to activate lower route
	    
	    #condSET := NOT (#i.status.vfbdeact OR #i.out.actmain OR #i.out.actupper OR #i.out.actlower) OR
	    NOT (#i.out.actmain OR #i.out.actupper OR #i.out.actlower) AND (#i.status.vfbmain OR #i.status.vfbupper OR #i.status.vfblower);
	    
	    "AFC_AlarmAckn"(trigger := NOT #i.status.vfblower AND #i.out.actlower,
	                    release := NOT #i.sim.lower AND #type = 1,
	                    ctrlpoint := FALSE,
	                    enackn := TRUE,
	                    ensiren := TRUE,
	                    p100ms := #p100ms,
	                    generalackn := #generalackn OR #i.faults.fpreset,
	                    reset := #reset OR #i.faults.fpreset,
	                    mute := #mute,
	                    delay := 0.0,
	                    plcackn => #faults.ctrl.plcackn_ftalower,
	                    alarm => #faults.ctrl.alarm_ftalower,
	                    siren => #faults.status.siren_ftalower,
	                    hmiackn := #faults.status.hmiackn_ftalower,
	                    Data := #i.faults.ftalower);
	    
	    //Network14: FAULT: Fail to deactivate
	    
	    #condSET := NOT (#i.status.vfbdeact OR #i.out.actmain OR #i.out.actupper OR #i.out.actlower) OR
	    NOT (#i.out.actmain OR #i.out.actupper OR #i.out.actlower) AND (#i.status.vfbmain OR #i.status.vfbupper OR #i.status.vfblower);
	    
	    "AFC_AlarmAckn"(trigger := #condSET,
	                    release := NOT #i.sim.deact,
	                    ctrlpoint := FALSE,
	                    enackn := TRUE,
	                    ensiren := TRUE,
	                    p100ms := #p100ms,
	                    generalackn := #generalackn OR #i.faults.fpreset,
	                    reset := #reset OR #i.faults.fpreset,
	                    mute := #mute,
	                    delay := 0.0,
	                    plcackn => #faults.ctrl.plcackn_ftd,
	                    alarm => #faults.ctrl.alarm_ftd,
	                    siren => #faults.status.siren_ftd,
	                    hmiackn := #faults.status.hmiackn_ftd,
	                    Data := #i.faults.ftd);
	    
	    //Network15: FAULT: Interlock violation
	    
	    #condSET := (#actmain AND #blockmain) OR (#actupper AND #blockupper) OR (#actlower AND #blocklower);
	    
	    "AFC_AlarmAckn"(trigger := #condSET,
	                    release := NOT (#i.status.ilactmain OR #i.status.ilactupper OR #i.status.ilactlower),
	                    ctrlpoint := FALSE,
	                    enackn := TRUE,
	                    ensiren := TRUE,
	                    p100ms := #p100ms,
	                    generalackn := #generalackn OR #i.faults.fpreset,
	                    reset := #reset OR #i.faults.fpreset,
	                    mute := #mute,
	                    delay := 0.0,
	                    plcackn => #faults.ctrl.plcackn_il,
	                    alarm => #faults.ctrl.alarm_il,
	                    siren => #faults.status.siren_il,
	                    hmiackn := #faults.status.hmiackn_il,
	                    Data := #i.faults.il);
	    
	END_REGION
	
	REGION STATUS  NW:16-21
	    
	    //Network16: STATUS: General Fault
	    
	    #i.status.fault := #i.faults.ftamain.status.alarm OR #i.faults.ftaupper.status.alarm OR #i.faults.ftalower.status.alarm OR #i.faults.ftd.status.alarm OR #i.faults.il.status.alarm;
	    
	    //Network17: STATUS: "Interlock activate main"
	    
	    #i.status.ilactmain := NOT (#blockmain OR #i.status.fault OR #i.out.actupper OR #i.out.actlower);
	    
	    //Network18: STATUS: "Interlock activate upper s/l"
	    
	    #i.status.ilactupper := NOT (#blockupper OR #i.status.fault OR #i.out.actmain OR #i.out.actlower);
	    
	    //Network19: STATUS: "Interlock activate lower s/l"
	    
	    #i.status.ilactlower := NOT (#blocklower OR #i.status.fault OR #i.out.actupper OR #i.out.actmain);
	    
	    //Network20: STATUS: Valve Graphic
	    
	    #i.status.icon := 0;
	    
	    IF #i.status.vfbmain AND #i.out.actmain AND NOT #i.status.fault
	    THEN
	        #i.status.icon := 1;
	    ELSIF #i.status.vfbupper AND #i.out.actupper AND NOT #i.status.fault
	    THEN
	        #i.status.icon := 2;
	    ELSIF #i.status.vfblower AND #i.out.actlower AND NOT #i.status.fault
	    THEN
	        #i.status.icon := 3;
	    ELSIF #i.status.fault AND #blink
	    THEN
	        #i.status.icon := 4;
	    END_IF;
	    
	    
	    //Network21: STATUS: Manual control buttons
	    
	    #i.ind.main := #i.man.main AND #i.ind.man;
	    #i.ind.upper := #i.man.upper AND #i.ind.upper;
	    #i.ind.lower := #i.man.lower AND #i.ind.lower;
	    #i.ind.deact := #i.ind.man AND NOT (#i.man.main OR #i.man.upper OR #i.man.lower);
	    
	END_REGION
	
	REGION OUTPUT NW: 22-24
	    
	    //Network22: OUTPUT: Activate main route
	    
	    #condSET := #i.man.main OR (#actmain AND #i.ind.auto);
	    #condRESET := NOT #i.status.ilactmain;
	    
	    "AFC_DelayONOFF"(cmd := #condSET,
	                     Pulse := #p100ms,
	                     Reset := #condRESET,
	                     on => #i.out.actmain,
	                     Data := #i.delaymain);
	    
	    //Network23: OUTPUT: Activate upper s/l route
	    
	    #condSET := #i.man.upper OR (#actupper AND #i.ind.auto);
	    #condRESET := #type = 1 OR NOT #i.status.ilactupper;
	    
	    "AFC_DelayONOFF"(cmd := #condSET,
	                     Pulse := #p100ms,
	                     Reset := #condRESET,
	                     on => #i.out.actupper,
	                     Data := #i.delayupper);
	    
	    //Network24: OUTPUT: Activate lower s/l route
	    
	    #condSET := #i.man.lower OR (#actlower AND #i.ind.auto);
	    #condRESET := #type = 1 OR NOT #i.status.ilactlower;
	    
	    "AFC_DelayONOFF"(cmd := #condSET,
	                     Pulse := #p100ms,
	                     Reset := #condRESET,
	                     on => #i.out.actlower,
	                     Data := #i.delaylower);
	    
	END_REGION
	
	REGION OUTPUT NW: 25
	    
	    //Network25: GEN: Move UDT outputs to FC outputs
	    
	    #main := #i.out.actmain;
	    #upper := #i.out.actupper;
	    #lower := #i.out.actlower;
	    #vfbmain := #i.status.vfbmain;
	    #vfbupper := #i.status.vfbupper;
	    #vfblower := #i.status.vfblower;
	    #vfbdeact := #i.status.vfbdeact;
	    
	END_REGION
	
	REGION BUTTON NW: 26
	    
	    //Network26: EXTRA: Button treatment
	    
	    IF #i.ind.auto THEN
	        #i.cmd.auto := FALSE;
	    END_IF;
	    
	    IF #i.ind.man THEN
	        #i.cmd.man := FALSE;
	    END_IF;
	    
	    IF #i.ind.main OR #i.ind.auto OR NOT #i.status.ilactmain THEN
	        #i.cmd.main := FALSE;
	    END_IF;
	    
	    IF #i.ind.upper OR #i.ind.auto OR NOT #i.status.ilactupper THEN
	        #i.cmd.upper := FALSE;
	    END_IF;
	    
	    IF #i.ind.lower OR #i.ind.auto OR NOT #i.status.ilactlower THEN
	        #i.cmd.lower := FALSE;
	    END_IF;
	    
	    IF #i.ind.deact OR #i.ind.auto THEN
	        #i.cmd.deact := FALSE;
	    END_IF;
	    
	    IF #i.status.fault THEN
	        #i.faults.fpreset := FALSE;
	    END_IF;
	    
	END_REGION
END_FUNCTION_BLOCK

FUNCTION_BLOCK "AFB_AlarmAckn"
TITLE = AFB_AlarmAckn
{ S7_Optimized_Access := 'TRUE' }
AUTHOR : CH
FAMILY : Aktina
NAME : Global
VERSION : 0.1
//AFB_AlarmAckn
   VAR_INPUT 
      trigger { ExternalAccessible := 'False'; ExternalVisible := 'False'; ExternalWritable := 'False'} : Bool;   // Alarm trigger
      release { ExternalAccessible := 'False'; ExternalVisible := 'False'; ExternalWritable := 'False'} : Bool;   // Release alarm
      ctrlpoint { ExternalAccessible := 'False'; ExternalVisible := 'False'; ExternalWritable := 'False'} : Bool;   // Control point (0=HMI, 1=PLC)
      enackn { ExternalAccessible := 'False'; ExternalVisible := 'False'; ExternalWritable := 'False'} : Bool;   // Enable acknowledgement (0=disable, 1=enable)
      ensiren { ExternalAccessible := 'False'; ExternalVisible := 'False'; ExternalWritable := 'False'} : Bool;   // Enable siren for this alarm
      p100ms { ExternalAccessible := 'False'; ExternalVisible := 'False'; ExternalWritable := 'False'} : Bool;   // 100ms pulse
      generalackn { ExternalAccessible := 'False'; ExternalVisible := 'False'; ExternalWritable := 'False'} : Bool;   // General acknowledgement
      reset { ExternalAccessible := 'False'; ExternalVisible := 'False'; ExternalWritable := 'False'} : Bool;   // Reset
      mute { ExternalAccessible := 'False'; ExternalVisible := 'False'; ExternalWritable := 'False'} : Bool;   // Mute siren
      delay { ExternalAccessible := 'False'; ExternalVisible := 'False'; ExternalWritable := 'False'} : Real;   // Delay on (s)
   END_VAR

   VAR_OUTPUT 
      plcackn { ExternalAccessible := 'False'; ExternalVisible := 'False'; ExternalWritable := 'False'} : Bool;   // PLC acknowledgement bit
      alarm { ExternalAccessible := 'False'; ExternalVisible := 'False'; ExternalWritable := 'False'} : Bool;   // Activation
      siren { ExternalAccessible := 'False'; ExternalVisible := 'False'; ExternalWritable := 'False'} : Bool;   // Siren
   END_VAR

   VAR_IN_OUT 
      hmiackn { ExternalAccessible := 'False'; ExternalVisible := 'False'; ExternalWritable := 'False'} : Bool;   // HMI acknowledgement bit
   END_VAR

   VAR RETAIN
      i : "UDT_ALARMACKN";   // Data processed in local memory
   END_VAR


BEGIN
	
	(*Calculate setpoint*)
	IF #ctrlpoint THEN
	    #i.setup."en" := #release;
	    #i.don.sp := REAL_TO_UINT(#delay * 10.0);
	ELSE
	    #i.don.sp := REAL_TO_UINT(#i.setup.spon * 10.0);
	END_IF;
	
	(*PLC acknowledgement*)
	IF #enackn AND #i.status.alarm THEN
	    IF (*#hmiackn OR*) #generalackn THEN
	        #i.status.plcackn := TRUE;
	    END_IF;
	ELSE
	    (*#hmiackn :=*) #i.status.plcackn := FALSE;
	END_IF;
	
	
	(*Reset counter*)
	IF NOT #trigger OR #i.status.alarm OR NOT #release OR NOT #i.setup."en" THEN
	    #i.don.actual := 0;
	END_IF;
	
	(*Alarming function*)
	IF #release AND #i.setup."en" THEN
	    
	    (*Count-up*)
	    #i.don.countup := #trigger AND #i.don.actual < #i.don.sp;
	    
	    IF #i.don.countup AND #p100ms AND NOT #i.don.end THEN
	        #i.don.actual := #i.don.actual + 1;
	    END_IF;
	    
	    (*Alarm & Siren generation*)
	    IF #trigger AND #i.don.actual >= #i.don.sp THEN
	        IF #ensiren AND NOT #i.status.alarm THEN
	            #i.status.siren := TRUE;
	        END_IF;
	        #i.status.alarm := TRUE;
	    END_IF;
	    
	    (*Siren reset*)
	    IF NOT #ensiren OR #mute OR #i.status.plcackn OR NOT #i.status.alarm THEN
	        #i.status.siren := FALSE;
	    END_IF;
	    
	    (*Alarm reset*)
	    IF NOT #trigger AND #i.status.alarm AND ((#enackn AND #i.status.plcackn) OR NOT #enackn) AND #reset THEN
	        #i.status.alarm := FALSE;
	    END_IF;
	    
	ELSE
	    #i.status.alarm := #i.status.siren := #i.don.countup := (*#hmiackn :=*) #i.status.plcackn := FALSE;
	END_IF;
	
	#plcackn := #i.status.plcackn;
	#alarm := #i.status.alarm;
	#siren := #i.status.siren;
	
	RETURN;
END_FUNCTION_BLOCK

FUNCTION_BLOCK "AFB_AlarmF"
{ S7_Optimized_Access := 'TRUE' }
VERSION : 0.1
   VAR_OUTPUT 
      faults : Struct
         pending : UDInt := 0;
         unackn : UDInt := 0;
      END_STRUCT;
      warnings : Struct
         pending { ExternalAccessible := 'False'; ExternalVisible := 'False'; ExternalWritable := 'False'} : UDInt := 0;   // False
         unackn { ExternalAccessible := 'False'; ExternalVisible := 'False'; ExternalWritable := 'False'} : UDInt := 0;   // False
      END_STRUCT;
      fault : Bool := false;
      warning : Bool := false;
      siren : Bool := false;
      icon : Byte := 16#0;
   END_VAR

   VAR 
      M_TYPE_FAULT : Array[0..#M_TYPES_FAULT] of Int := ["M_ADIN", "M_AIN", "M_DIFF", "M_DIN", "M_MTR", "M_MTRLIN", "M_MTRDIR", "M_VLV", "M_PLANT"];
      M_TYPE_WARNING : Array[0..#M_TYPES_WARNING] of Int := ["M_AIN", "M_DIFF", "M_PLANT"];
      nFault : Struct
         Alarm : Array[0..#M_TYPES_FAULT] of UDInt;
         Ackn : Array[0..#M_TYPES_FAULT] of UDInt;
         Siren : Array[0..#M_TYPES_FAULT] of UDInt;
      END_STRUCT;
      nWarning : Struct
         Alarm : Array[0..#M_TYPES_WARNING] of UDInt;
         Ackn : Array[0..#M_TYPES_WARNING] of UDInt;
         Siren : Array[0..#M_TYPES_WARNING] of UDInt;
      END_STRUCT;
   END_VAR

   VAR_TEMP 
      i : Int;
      totalFault : Struct
         alarm : UDInt;
         ackn : UDInt;
         siren : UDInt;
      END_STRUCT;
      totalWarning : Struct
         alarm : UDInt;
         ackn : UDInt;
         siren : UDInt;
      END_STRUCT;
   END_VAR

   VAR CONSTANT 
      tADIN : Int := 0;
      tAIN : Int := 1;
      tDIFF : Int := 2;
      tDIN : Int := 3;
      tMTR : Int := 4;
      tMTRLIN : Int := 5;
      tMTRDIR : Int := 6;
      tVLV : Int := 7;
      tPLANT : Int := 8;
      wAIN : Int := 0;
      wDIFF : Int := 1;
      wPLANT : Int := 2;
      M_TYPES_FAULT : Int := 8;
      M_TYPES_WARNING : Int := 2;
   END_VAR


BEGIN
	REGION Custom faults
	     "iPALARMS"();
	     
	     END_REGION Custom faults
	
	REGION FAULTS
	    
	    #totalFault.alarm := 0;
	    #totalFault.ackn := 0;
	    #totalFault.siren := 0;
	    
	    // Set number of instances for the statistics calculations
	    #M_TYPE_FAULT[#tADIN] := "M_ADIN";
	    #M_TYPE_FAULT[#tAIN] := "M_AIN";
	    #M_TYPE_FAULT[#tDIFF] := "M_DIFF";
	    #M_TYPE_FAULT[#tDIN] := "M_DIN";
	    #M_TYPE_FAULT[#tMTR] := "M_MTR";
	    #M_TYPE_FAULT[#tMTRLIN] := "M_MTRLIN";
	    #M_TYPE_FAULT[#tMTRDIR] := "M_MTRDIR";
	    #M_TYPE_FAULT[#tVLV] := "M_VLV";
	    #M_TYPE_FAULT[#tPLANT] := "M_PLANT";
	    
	    #M_TYPE_WARNING[#wAIN] := "M_AIN";
	    #M_TYPE_WARNING[#wDIFF] := "M_DIFF";
	    #M_TYPE_WARNING[#wPLANT] := "M_PLANT";
	    
	    
	    
	    FOR #i := #tADIN TO #tPLANT DO
	        
	        "AFC_AlarmTypeStatistics"(TYPE := #i,
	                                  M_TYPE := #M_TYPE_FAULT[#i],
	                                  nAlarm => #nFault.Alarm[#i],
	                                  nAckn => #nFault.Ackn[#i],
	                                  nSiren => #nFault.Siren[#i]);
	        
	        #totalFault.alarm := #totalFault.alarm + #nFault.Alarm[#i];
	        #totalFault.ackn := #totalFault.ackn + #nFault.Ackn[#i];
	        #totalFault.siren := #totalFault.siren + #nFault.Siren[#i];
	        
	    END_FOR;
	    
	END_REGION
	
	REGION WARNINGS
	    
	    #totalWarning.alarm := 0;
	    #totalWarning.ackn := 0;
	    #totalWarning.siren := 0;
	    
	    FOR #i := #wAIN TO #wPLANT DO
	        
	        "AFC_WarnTypeStatistics"(TYPE := #i,
	       M_TYPE := #M_TYPE_WARNING[#i],
	       nAlarm => #nWarning.Alarm[#i],
	       nAckn => #nWarning.Ackn[#i],
	       nSiren => #nWarning.Siren[#i]);
	        
	        #totalWarning.alarm := #totalWarning.alarm + #nWarning.Alarm[#i];
	        #totalWarning.ackn := #totalWarning.ackn + #nWarning.Ackn[#i];
	        #totalWarning.siren := #totalWarning.siren + #nWarning.Siren[#i];
	        
	    END_FOR;
	    
	    
	END_REGION
	
	(*Siren*)
	
	#faults.pending := #totalFault.alarm;
	#faults.unackn := #totalFault.alarm + #totalFault.ackn;
	
	#warnings.pending := #totalWarning.alarm;
	#warnings.unackn := #totalWarning.alarm + #totalWarning.ackn;
	
	#fault := #totalFault.alarm <> 0;
	#warning := #totalWarning.alarm <> 0;
	#siren := #totalFault.siren <> 0 OR #totalWarning.siren <> 0;
	
	(*Icon*)
	IF (#totalFault.alarm <> 0)
	THEN
	    #icon := 4;
	    
	ELSIF (#totalWarning.alarm <> 0)
	THEN
	    #icon := 2;
	    
	ELSE
	    #icon := 1;
	END_IF;
END_FUNCTION_BLOCK

FUNCTION "AFC_AlarmTypeStatistics" : Void
{ S7_Optimized_Access := 'TRUE' }
VERSION : 0.1
   VAR_INPUT 
      "TYPE" : Int;
      M_TYPE : Int;
   END_VAR

   VAR_OUTPUT 
      nAlarm : UDInt;
      nAckn : UDInt;
      nSiren : UDInt;
   END_VAR

   VAR_TEMP 
      i : Int;
      alarm : Word;
      ackn : Word;
      siren : Word;
   END_VAR

   VAR CONSTANT 
      tADIN : Int := 0;
      tAIN : Int := 1;
      tDIFF : Int := 2;
      tDIN : Int := 3;
      tMTR : Int := 4;
      tMTRLIN : Int := 5;
      tMTRDIR : Int := 6;
      tVLV : Int := 7;
      tPLANT : Int := 8;
   END_VAR


BEGIN
	#nAlarm := 0;
	#nAckn := 0;
	#nSiren := 0;
	
	FOR #i := 0 TO #M_TYPE DO
	    
	    CASE #TYPE OF
	        #tADIN:
	             
	             "AFC_AlarmGatherArray"(
	                                    ctrl := "FAULTS".ADIN[#i].ctrl,
	                                    status := "FAULTS".ADIN[#i].status,
	                                    _ctrl => #alarm,
	                                    _status => #ackn);
	                  
	        #tAIN:
	            
	             "AFC_AlarmGatherStruct"(
	                              ctrl := "FAULTS".AIN[#i].ctrl,
	                              status := "FAULTS".AIN[#i].status,
	                              _ctrl => #alarm,
	                              _status => #ackn);
	            
	        #tDIFF:
	            
	             "AFC_AlarmGatherStruct"(
	                              ctrl := "FAULTS".DIFF[#i].ctrl,
	                              status := "FAULTS".DIFF[#i].status,
	                              _ctrl => #alarm,
	                              _status => #ackn);
	            
	        #tDIN:
	            
	             "AFC_AlarmGatherArray"(
	                              ctrl := "FAULTS".DIN[#i].ctrl,
	                              status := "FAULTS".DIN[#i].status,
	                              _ctrl => #alarm,
	                              _status => #ackn);
	            
	        #tMTR:
	            
	             "AFC_AlarmGatherStruct"(
	                              ctrl := "FAULTS".MTR[#i].ctrl,
	                              status := "FAULTS".MTR[#i].status,
	                              _ctrl => #alarm,
	                              _status => #ackn);
	            
	        #tMTRLIN:
	            
	             "AFC_AlarmGatherStruct"(
	                              ctrl := "FAULTS".MTRLIN[#i].ctrl,
	                              status := "FAULTS".MTRLIN[#i].status,
	                              _ctrl => #alarm,
	                              _status => #ackn);
	            
	        #tMTRDIR:
	            
	             "AFC_AlarmGatherStruct"(
	                              ctrl := "FAULTS".MTRDIR[#i].ctrl,
	                              status := "FAULTS".MTRDIR[#i].status,
	                              _ctrl => #alarm,
	                              _status => #ackn);
	            
	        #tVLV:
	            
	             "AFC_AlarmGatherStruct"(
	                              ctrl := "FAULTS".VLV[#i].ctrl,
	                              status := "FAULTS".VLV[#i].status,
	                              _ctrl => #alarm,
	                              _status => #ackn);
	            
	       #tPLANT:
	            
	            "AFC_AlarmGatherArray"(
	                              ctrl := "FAULTS".Plant[#i].ctrl,
	                              status := "FAULTS".Plant[#i].status,
	                              _ctrl => #alarm,
	                              _status => #ackn);
	            
	        ELSE  // Statement section ELSE
	            ;
	    END_CASE;
	    
	    
	    #nAlarm := #nAlarm + "countAlarms"(#alarm.%B0);
	    #nAckn := #nAckn + "countAlarms"(#ackn.%B1);
	    #nSiren := #nSiren + "countAlarms"(#ackn.%B0);
	    
	    
	END_FOR;
	
	
END_FUNCTION

FUNCTION "AFC_AlarmGatherArray" : Void
{ S7_Optimized_Access := 'TRUE' }
VERSION : 0.1
   VAR_INPUT 
      ctrl : Array[0..15] of Bool;   // External data (Primary fault data - alarm & plc ackn)
      status : Array[0..15] of Bool;   // External data (Secondary fault data - siren & hmi ackn)
   END_VAR

   VAR_OUTPUT 
      _ctrl : Word;
      _status : Word;
   END_VAR

   VAR_TEMP 
      tCtrl : Struct
         bit8 : Bool;
         bit9 : Bool;
         bit10 : Bool;
         bit11 : Bool;
         bit12 : Bool;
         bit13 : Bool;
         bit14 : Bool;
         bit15 : Bool;
         bit0 : Bool;
         bit1 : Bool;
         bit2 : Bool;
         bit3 : Bool;
         bit4 : Bool;
         bit5 : Bool;
         bit6 : Bool;
         bit7 : Bool;
      END_STRUCT;
      tStatus : Struct
         bit8 : Bool;
         bit9 : Bool;
         bit10 : Bool;
         bit11 : Bool;
         bit12 : Bool;
         bit13 : Bool;
         bit14 : Bool;
         bit15 : Bool;
         bit0 : Bool;
         bit1 : Bool;
         bit2 : Bool;
         bit3 : Bool;
         bit4 : Bool;
         bit5 : Bool;
         bit6 : Bool;
         bit7 : Bool;
      END_STRUCT;
   END_VAR


BEGIN
	
	    GATHER(IN := #ctrl,
	           OUT => #_ctrl);
	    GATHER(IN := #status,
	           OUT => #_status);
	    
END_FUNCTION

FUNCTION "AFC_AlarmGatherStruct" : Void
{ S7_Optimized_Access := 'TRUE' }
VERSION : 0.1
   VAR_INPUT 
      ctrl : Struct   // External data (Primary fault data - alarm & plc ackn)
         bit8 : Bool;
         bit9 : Bool;
         bit10 : Bool;
         bit11 : Bool;
         bit12 : Bool;
         bit13 : Bool;
         bit14 : Bool;
         bit15 : Bool;
         bit0 : Bool;
         bit1 : Bool;
         bit2 : Bool;
         bit3 : Bool;
         bit4 : Bool;
         bit5 : Bool;
         bit6 : Bool;
         bit7 : Bool;
      END_STRUCT;
      status : Struct   // External data (Secondary fault data - siren & hmi ackn)
         bit8 : Bool;
         bit9 : Bool;
         bit10 : Bool;
         bit11 : Bool;
         bit12 : Bool;
         bit13 : Bool;
         bit14 : Bool;
         bit15 : Bool;
         bit0 : Bool;
         bit1 : Bool;
         bit2 : Bool;
         bit3 : Bool;
         bit4 : Bool;
         bit5 : Bool;
         bit6 : Bool;
         bit7 : Bool;
      END_STRUCT;
   END_VAR

   VAR_OUTPUT 
      _ctrl : Word;
      _status : Word;
   END_VAR


BEGIN
	
	    GATHER(IN := #ctrl,
	           OUT => #_ctrl);
	    GATHER(IN := #status,
	           OUT => #_status);
	    
END_FUNCTION

FUNCTION "countAlarms" : UDInt
{ S7_Optimized_Access := 'TRUE' }
VERSION : 0.1
   VAR_INPUT 
      byteIn : Byte;
   END_VAR

   VAR_TEMP 
      i : UDInt;
      count : UDInt;
   END_VAR

   VAR CONSTANT 
      ONE : Word := 16#1;
   END_VAR


BEGIN
	FOR #i := 0 TO 7 DO
	    
	    IF (#byteIn AND SHL(IN := #ONE, N := #i)) <> 0 THEN
	        
	        #count := #count + 1;
	        
	    END_IF;
	    
	END_FOR;
	
	#countAlarms := #count;
END_FUNCTION

FUNCTION "AFC_WarnTypeStatistics" : Void
{ S7_Optimized_Access := 'TRUE' }
VERSION : 0.1
   VAR_INPUT 
      "TYPE" : Int;
      M_TYPE : Int;
   END_VAR

   VAR_OUTPUT 
      nAlarm : UDInt;
      nAckn : UDInt;
      nSiren : UDInt;
   END_VAR

   VAR_TEMP 
      i : Int;
      alarm : Word;
      ackn : Word;
      siren : Word;
   END_VAR

   VAR CONSTANT 
      wDIFF : Int := 1;
      wAIN : Int := 0;
      wPLANT : Int := 2;
   END_VAR


BEGIN
	#nAlarm := 0;
	#nAckn := 0;
	#nSiren := 0;
	
	FOR #i := 0 TO #M_TYPE DO
	    
	    CASE #TYPE OF
	         #wAIN:
	              
	              "AFC_AlarmGatherStruct"(
	                                ctrl := "WARNINGS".AIN[#i].ctrl,
	                                status := "WARNINGS".AIN[#i].status,
	                                _ctrl => #alarm,
	                                _status => #ackn);
	              
	         #wDIFF:
	            
	             "AFC_AlarmGatherStruct"(
	                              ctrl:="WARNINGS".DIFF[#i].ctrl,
	                              status:="WARNINGS".DIFF[#i].status,
	                              _ctrl=>#alarm,
	                              _status=>#ackn);
	            
	       #wPLANT:
	            
	            "AFC_AlarmGatherArray"(
	                              ctrl := "WARNINGS".Plant[#i].ctrl,
	                              status := "WARNINGS".Plant[#i].status,
	                              _ctrl => #alarm,
	                              _status => #ackn);
	            
	        ELSE  // Statement section ELSE
	            ;
	    END_CASE;
	    
	    
	    #nAlarm := #nAlarm + "countAlarms"(#alarm.%B0);
	    #nAckn := #nAckn + "countAlarms"(#ackn.%B1);
	    #nSiren := #nSiren + "countAlarms"(#ackn.%B0);
	    
	END_FOR;
	
	
END_FUNCTION

FUNCTION_BLOCK "AFB_AlarmGroup"
TITLE = AFB_AlarmGroup
{ S7_Optimized_Access := 'TRUE' }
AUTHOR : CH
FAMILY : Aktina
NAME : Global
VERSION : 0.1
//AFB_AlarmGroup
   VAR_INPUT 
      req : Bool;   // Request
      "db" : DB_ANY;   // DB with the alarm data
   END_VAR

   VAR_OUTPUT 
      ret_val : Int;   // Return value (256=wrong DB structure, <>256=attr_db ret_val)
   END_VAR

   VAR_IN_OUT 
      alarm : Bool;   // New alarm
      siren : Bool;   // Siren
      pending : UDInt;   // Pending alarms
      unackn : UDInt;   // Uacknowledged alarms
   END_VAR

   VAR 
      attr : Struct   // DB attributes
         ret_val : Int;
         length : UDInt;
         attrib : Byte;
      END_STRUCT;
      cond : Struct   // Conditions
         siren : Bool;   // There is a siren bit enabled
         alarm : Bool;   // There is a pending alarm
         unackn : Bool;   // There is an unacknowledged alarm
      END_STRUCT;
      peek : Struct   // Peek data
         offset : DInt;   // Memory offset for peek instruction starting byte
         memory : Byte;   // Memory returned by peek instruction
      END_STRUCT;
      alarms : Struct   // Alarms number
         pending : UDInt;   // Pending alarms
         siren : UDInt;   // Siren requestsnumber
         ackn : UDInt;   // Acknowledged alarms
         unackn : UDInt;   // Uacknowledged alarms
      END_STRUCT;
      temp : Struct   // Temporary memory examined
         pending : Byte;   // Pending alarm memory
         ackn : Byte;   // Acknowledged alarm memory
         siren : Byte;   // Siren memory
      END_STRUCT;
      groups : UInt;   // Groups number
      n : UInt;   // Operand n
      x : Byte;   // Operand x
   END_VAR


BEGIN
	
	REGION Group monitoring
	    
	IF #req THEN
	    
	    #attr.ret_val := ATTR_DB(REQ := #req, DB_NUMBER := #db, DB_LENGTH => #attr.length, ATTRIB => #attr.attrib);
	    
	    #groups := UDINT_TO_UINT(#attr.length / 4);
	    
	    IF (UDINT_TO_UINT(#attr.length) - (#groups * 4)) <> 0 OR #attr.length = 0 THEN
	        #ret_val := 256;
	        #alarm := #siren := FALSE;
	        #alarms.unackn := #alarms.pending := #alarms.ackn := 0;
	        
	        RETURN;
	        
	    ELSE
	        #ret_val := #attr.ret_val;
	    END_IF;
	    
	(*Check for pending and unacknowledged alarms.
	If there is no pending alarm then we do not continue and check for siren.
	The software is optimised to check for all in the min possible execution time.*)
	    
	(*Alarms*)
	    #n := 0;
	    #alarms.pending := #alarms.ackn := #alarms.siren := 0;
	    WHILE #n < #groups DO
	        
	        #peek.offset := 0 + #n * 4;
	        
	        #peek.memory := PEEK(area := 16#84, dbNumber := #db, byteOffset := #peek.offset);
	        
	        IF #peek.memory <> 0 THEN // We are checking only if byte is full
	            
	            #temp.pending := #peek.memory;
	            
	            #peek.offset := 1 + #n * 4; // Check also for acknowledged alarms
	            
	            #peek.memory := PEEK(area := 16#84, dbNumber := #db, byteOffset := #peek.offset);
	            
	            #temp.ackn := #peek.memory;
	            
	            #peek.offset := 2 + #n * 4; // Check also for acknowledged alarms
	            
	            #peek.memory := PEEK(area := 16#84, dbNumber := #db, byteOffset := #peek.offset);
	            
	            #temp.siren := #peek.memory;
	            
	            WHILE #temp.pending <> 0 DO
	                IF (#temp.pending AND 16#1) <> 0 THEN // Check for pending alarms
	                    #alarms.pending := #alarms.pending + 1;
	                    IF (#temp.ackn AND 16#1) <> 0 THEN // Check for acknowledged alarms
	                        #alarms.ackn := #alarms.ackn + 1;
	                    END_IF;
	                    IF (#temp.siren AND 16#1) <> 0 THEN // Check for siren requests
	                        #alarms.siren := #alarms.siren + 1;
	                    END_IF;
	                END_IF;
	                #temp.pending := SHR_BYTE(IN := #temp.pending, N := 1);
	                #temp.ackn := SHR_BYTE(IN := #temp.ackn, N := 1);
	                #temp.siren := SHR_BYTE(IN := #temp.siren, N := 1);
	            END_WHILE;
	            
	        ELSE
	            
	            #temp.pending := #temp.ackn := #temp.siren := #peek.memory := 0;
	            
	        END_IF;
	        #n := #n + 1;
	    END_WHILE;
	    
	    #alarms.unackn := #alarms.pending - #alarms.ackn; // Unacknowledged alarms number
	    
	    #cond.alarm := #alarms.pending <> 0; // Condition for pending alarms
	    #cond.siren := #alarms.siren <> 0; // Condition for siren
	    
	ELSE
	   
	    #ret_val := 0;
	    #cond.alarm := #cond.siren := FALSE;
	    #alarms.unackn := #alarms.pending := #alarms.ackn := 0;
	    
	END_IF;
	
	END_REGION Group monitoring
	
	REGION Output
	    // We alter the output only if it is necessary
	    
	    IF (#cond.alarm = TRUE) THEN
	        #alarm := TRUE;
	    END_IF;
	    
	    IF (#cond.siren = TRUE) THEN
	        #siren := TRUE;
	    END_IF;
	    
	    #pending := #alarms.pending;
	    #unackn := #alarms.unackn;
	    
	    END_REGION Output
	
	
	RETURN;
	    
END_FUNCTION_BLOCK

FUNCTION "AFC_Array_To_Word" : Void
TITLE = AFC_Array_To_Word
{ S7_Optimized_Access := 'FALSE' }
AUTHOR : CH
FAMILY : Aktina
NAME : Global
VERSION : 0.1
//AFC_Array_To_Word
   VAR_INPUT 
      s : Array[0..15] of Bool;
   END_VAR

   VAR_OUTPUT 
      w : Word;
   END_VAR

   VAR_TEMP 
      ts : Array[0..15] of Bool;
      tw AT ts : Word;
   END_VAR


BEGIN
	#ts := #s;
	
	#w := #tw;
	
	#tw := 0;
	
	RETURN;
END_FUNCTION

FUNCTION "AFC_Struct_To_Word" : Void
TITLE = AFC_Struct_To_Word
{ S7_Optimized_Access := 'FALSE' }
AUTHOR : CH
FAMILY : Aktina
NAME : Global
VERSION : 0.1
//AFC_Struct_To_Word
   VAR_INPUT 
      s : Struct
         bit0 : Bool;
         bit1 : Bool;
         bit2 : Bool;
         bit3 : Bool;
         bit4 : Bool;
         bit5 : Bool;
         bit6 : Bool;
         bit7 : Bool;
         bit8 : Bool;
         bit9 : Bool;
         bit10 : Bool;
         bit11 : Bool;
         bit12 : Bool;
         bit13 : Bool;
         bit14 : Bool;
         bit15 : Bool;
      END_STRUCT;
   END_VAR

   VAR_OUTPUT 
      w : Word;
   END_VAR

   VAR_TEMP 
      ts : Struct
         bit0 : Bool;
         bit1 : Bool;
         bit2 : Bool;
         bit3 : Bool;
         bit4 : Bool;
         bit5 : Bool;
         bit6 : Bool;
         bit7 : Bool;
         bit8 : Bool;
         bit9 : Bool;
         bit10 : Bool;
         bit11 : Bool;
         bit12 : Bool;
         bit13 : Bool;
         bit14 : Bool;
         bit15 : Bool;
      END_STRUCT;
      tw AT ts : Word;
   END_VAR


BEGIN
	#ts := #s;
	
	#w := #tw;
	
	#tw := 0;
	
	RETURN;
END_FUNCTION

FUNCTION "AFC_Word_To_Array" : Void
TITLE = AFC_Word_To_Array
{ S7_Optimized_Access := 'FALSE' }
AUTHOR : CH
FAMILY : Aktina
NAME : Global
VERSION : 0.1
//AFC_Word_To_Array
   VAR_INPUT 
      w : Word;
   END_VAR

   VAR_OUTPUT 
      s : Array[0..15] of Bool;
   END_VAR

   VAR_TEMP 
      tw : Word;
      ts AT tw : Array[0..15] of Bool;
   END_VAR


BEGIN
	#tw := #w;
	
	#s := #ts;
	
	#tw := 16#0;
	
	RETURN;
END_FUNCTION

FUNCTION "AFC_Word_To_Struct" : Void
TITLE = AFC_Word_to_Struct
{ S7_Optimized_Access := 'FALSE' }
AUTHOR : CH
FAMILY : Aktina
NAME : Global
VERSION : 0.1
//AFC_Word_to_Struct
   VAR_INPUT 
      w : Word;
   END_VAR

   VAR_OUTPUT 
      s : Struct
         bit0 : Bool;
         bit1 : Bool;
         bit2 : Bool;
         bit3 : Bool;
         bit4 : Bool;
         bit5 : Bool;
         bit6 : Bool;
         bit7 : Bool;
         bit8 : Bool;
         bit9 : Bool;
         bit10 : Bool;
         bit11 : Bool;
         bit12 : Bool;
         bit13 : Bool;
         bit14 : Bool;
         bit15 : Bool;
      END_STRUCT;
   END_VAR

   VAR_TEMP 
      tw : Word;
      ts AT tw : Struct
         bit0 : Bool;
         bit1 : Bool;
         bit2 : Bool;
         bit3 : Bool;
         bit4 : Bool;
         bit5 : Bool;
         bit6 : Bool;
         bit7 : Bool;
         bit8 : Bool;
         bit9 : Bool;
         bit10 : Bool;
         bit11 : Bool;
         bit12 : Bool;
         bit13 : Bool;
         bit14 : Bool;
         bit15 : Bool;
      END_STRUCT;
   END_VAR


BEGIN
	#tw := #w;
	
	#s := #ts;
	
	#tw := 16#0;
	
	RETURN;
END_FUNCTION

FUNCTION_BLOCK "libGeo_TankV_1"
TITLE = libGeo_TankV
{ S7_Optimized_Access := 'TRUE' }
AUTHOR : CH
FAMILY : Aktina
NAME : Geometry
VERSION : 0.1
//Half cone base tank mass calculation.
//The calculation is based on the principle that by pressure we always get the height of a media with ρ=1 (equal to water). From that we can calculate the volume using the tank dimensions. So we know for a ρ=1 media the volume and by that the mass. So for every ther media no matter the ρ value we know the mass based on the fact that the pressure would be the same. The volume can then be calculated if we know the ρ.
   VAR_INPUT 
      r { ExternalAccessible := 'False'; ExternalVisible := 'False'; ExternalWritable := 'False'} : Real;   //  Media density
      d { ExternalAccessible := 'False'; ExternalVisible := 'False'; ExternalWritable := 'False'} : Real;   //  Tank diameter
      hPt { ExternalAccessible := 'False'; ExternalVisible := 'False'; ExternalWritable := 'False'} : Real;   //  Pressure transmitter installation height
      hBase { ExternalAccessible := 'False'; ExternalVisible := 'False'; ExternalWritable := 'False'} : Real;   //  Base height
      hCyl { ExternalAccessible := 'False'; ExternalVisible := 'False'; ExternalWritable := 'False'} : Real;   //  Cylinder height
      hAct { ExternalAccessible := 'False'; ExternalVisible := 'False'; ExternalWritable := 'False'} : Real;   //  Actual measured height
   END_VAR

   VAR_OUTPUT 
      mass : Real;   //  Media mass
      vol : Real;   //  Media volume
      height : Real;   //  Media height
   END_VAR

   VAR 
      statHTrue : Real;   //  Static value for the true height of the media inside the tank
      statVol : Real;   //  Static value for the volume of the media inside the tank
   END_VAR

   VAR_TEMP 
      tempHZn1 : Real;   //  Temporary value for the height of media inside the first zone of the tank, the base
      tempHZn2 : Real;   //  Temporary value for the height of media inside the second zone of the tank, the cylinder
   END_VAR

   VAR CONSTANT 
      pi : Real := 3.14159;
   END_VAR


BEGIN
	REGION BLOCK HEADER
	    //===============================================================================
	    // CH / (c)Copyright (2021)
	    //-------------------------------------------------------------------------------
	    // Title:               (Volume calculation of water tank)
	    // Comment/Function:    ()
	    // Library/Family:      (Aktina/Tools/Geometry)
	    // Author:              (CH)
	    // Tested with:         (V17)
	    // Engineering:         (TIA Step7 Professional V17)
	    // Restrictions:        ()
	    // Requirements:        (S7 CPUs)
	    // Memory access:       (Optimized)
	    // Notes:             
	    //-------------------------------------------------------------------------------
	    // Change log table:
	    // Version  | Date       | Dev in charge          | Changes
	    //----------|------------|------------------------|------------------------------
	    // 01.00.00 | 2022-05-18 | (CH)                   | First released version
	    //===============================================================================
	END_REGION
	
	REGION BLOCK NOTES
	    //===============================================================================
	    // 1:Half cone base tank mass calculation.
	    // The calculation is based on The principle that by pressure we always get the height of
	    // a media with ρ=1 (equal to water). From that we can calculate the volume using the tank
	    // dimensions. So we know for a ρ=1 media the volume and by that the #mass.
	    // So for every ther media no matter the ρ value we know the mass based on the fact that
	    // the pressure would be the same. The volume can then be calculated if we know the ρ.
	    //===============================================================================
	END_REGION
	
	REGION CALCULATION
	    // Actual height calculation due to the offset height of the transmitter
	    #statHTrue := #hAct + #hPt;
	    
	    // Null volume and stop if the height of media is below the transmitter
	    IF #hAct <= 1.0 THEN
	        #statHTrue := 0;
	        #statVol := 0;
	        
	        #height := #statHTrue;
	        #mass := #statVol;
	        #vol := #statVol / #r;
	        
	        ENO := TRUE;
	        
	        RETURN;
	        
	        
	        
	    END_IF;
	    
	    // Height in base
	    IF #statHTrue < #hBase  THEN
	        #tempHZn1 := #statHTrue;
	    ELSE
	        #tempHZn1 := #hBase;
	    END_IF;
	    
	    // Height in cylinder
	    IF #statHTrue <= #hBase THEN
	        #tempHZn2 := 0.0;
	    ELSIF #statHTrue >= (#hBase + #hCyl) THEN
	        #tempHZn2 := #hCyl;
	    ELSE
	        #tempHZn2 := #statHTrue - #hBase;
	        END_IF;
	        
	    // Volume calculation
	        #statVol := (#pi * SQR_REAL(#d) * (#tempHZn1)) / 8 + (#pi * SQR_REAL(#d) * (#tempHZn2)) / 4;
	        
	        #height := #tempHZn1 + #tempHZn2;
	        #mass := #statVol;
	        #vol := #statVol / #r;
	        
	        ENO := TRUE;
	        
	END_REGION
END_FUNCTION_BLOCK

FUNCTION_BLOCK "AFB_ExpSmooth_v2"
TITLE = AFB_ExpSmooth_v2
{ S7_Optimized_Access := 'TRUE' }
AUTHOR : CH
FAMILY : Aktina
NAME : Global
VERSION : 0.1
//AFB_ExpSmooth_v2
   VAR_INPUT 
      In { ExternalAccessible := 'False'; ExternalVisible := 'False'; ExternalWritable := 'False'} : Real;   // Real to be smoothed
      p1s : Bool;   // Pulse for 1 s
      reset : Bool;   // Reset faults
      t_sys {InstructionName := 'DTL'; LibVersion := '1.0'; ExternalAccessible := 'False'; ExternalVisible := 'False'; ExternalWritable := 'False'} : DTL;   // System time
   END_VAR

   VAR_OUTPUT 
      Out { ExternalAccessible := 'False'; ExternalVisible := 'False'; ExternalWritable := 'False'} : Real;   // Scaled Value
   END_VAR

   VAR RETAIN
      i : "UDT_EXPSM";   // UDT containing faceplate data
      exp : Struct   // Exponential smoothing operands
         init : Bool;   // Initialization routine
         Sn : Real;   // Sn = n - output of smoothing
         Xn : Real;   // Xn = n - sample of analog value
         lim_up : Real;   // Limit up
         lim_down : Real;   // Limit down
         t_buf {InstructionName := 'DTL'; LibVersion := '1.0'} : DTL;   // Time buffering from last call of the function
         t_diff : Bool;   // t_diff = t_sys - t_buf (Ltime, ns)
      END_STRUCT;
   END_VAR
   VAR 
      err : Int;
      startob_si {InstructionName := 'SI_classic'; LibVersion := '1.0'; S7_SetPoint := 'False'} : SI_classic;
      lastob_si {InstructionName := 'SI_classic'; LibVersion := '1.0'; S7_SetPoint := 'False'} : SI_classic;
      logical1 { ExternalAccessible := 'False'; ExternalVisible := 'False'; ExternalWritable := 'False'} : Bool;
   END_VAR


BEGIN
	// Import value
	#i.actual := #In;
	
	// Check if smoothing is enabled
	IF #i.exp_sm AND NOT #i.simcmd THEN
	    
	    // Check system
	    #err := RD_SINFO(TOP_SI => #lastob_si, START_UP_SI => #startob_si);
	    
	    // Init routine
	    IF #lastob_si.EV_NUM = 1 OR #lastob_si.EV_NUM = 2 OR #lastob_si.EV_NUM = 4 THEN
	        #exp.init := false;
	    END_IF;
	    
	    // Enter routine
	    #exp.Xn := #i.actual;
	    #exp.lim_up := #exp.Xn + #i.limit;
	    #exp.lim_down := #exp.Xn - #i.limit;
	    
	   // #exp.t_diff := T_DIFF(IN1 := #t_sys, IN2 := #exp.t_buf);
	    //#i.dt := UDINT_TO_REAL(LTIME_TO_UDINT(#exp.t_diff)) / 1000000.0;
	    
	    IF #i.T <= 0 THEN // Force the period to be higher than 0 to avoid infinity on the exponent
	        #i.T := #i.dt / 1000.0;
	    END_IF;
	    
	    IF #i.dt > 0 AND #i.T > #i.dt / 1000.0 THEN
	        #i.a := 1 - EXP(- #i.dt / (1000.0 * #i.T));
	    END_IF;
	    
	(* startup initialisation *)
	    IF NOT #exp.init OR #i.a <= 0 OR #i.a >= 1 THEN
	        #exp.init := TRUE;
	        #exp.Sn := #exp.Xn;
	    ELSIF #exp.Sn >= #exp.lim_down AND #exp.Sn <= #exp.lim_up THEN
	        #exp.Sn := #exp.Xn;
	    ELSE
	        #exp.Sn := #exp.Sn + (#exp.Xn - #exp.Sn) * #i.a;
	    END_IF;
	    
	ELSIF #i.simcmd THEN
	    #exp.init := false;
	    #exp.Xn := #i.actual;
	    #exp.Sn := #i.simvalue;
	ELSE
	    #exp.init := false;
	    #exp.Xn := #i.actual;
	    #exp.Sn := #i.actual;
	        
	END_IF;
	
	// Buffering
	#exp.t_buf := #t_sys;
	#i.output := #exp.Sn;
	
	RETURN;
	
	
END_FUNCTION_BLOCK

FUNCTION_BLOCK "libMath_Total64REAL"
TITLE = libMath_Total64REAL
{ S7_Optimized_Access := 'TRUE' }
AUTHOR : CH
FAMILY : Aktina
NAME : MATH
VERSION : 1.0
//libMath_Total64REAL
   VAR_INPUT 
      pulse { ExternalAccessible := 'False'; ExternalVisible := 'False'; ExternalWritable := 'False'} : Bool;   //  TRUE: Add preset quantity to the totalizer
      refresh : Bool;   //  TRUE: Refresh calculation of analytical preset number
   END_VAR

   VAR_IN_OUT 
      "dt" : "typeTotal64REAL";   //  Totalizer's data
   END_VAR

   VAR 
      statPulseOld { ExternalWritable := 'False'} : Bool;   //  Static value for 'pulse' input used for edge detection
      statValid { ExternalWritable := 'False'} : Bool;   //  Static value for validating the preset conversion
      statTotalInt { ExternalWritable := 'False'} : DInt;   //  Static value for the integer part of 'statTotal'
      statTotalDec { ExternalWritable := 'False'} : DInt;   //  Static value for the decimal part of the 'statTotal'
      statExp { ExternalWritable := 'False'} : DInt;   //  Static value for the power of 10 calculated by 10^precision
      statTotal { ExternalWritable := 'False'} : LReal;   //  Static value for the 'total' output
      statPreset { ExternalWritable := 'False'} : Real := 0.0;   //  Static value for the 'setup.preset' input
      statPrecision { ExternalWritable := 'False'} : USInt;   //  Static value for the 'setup.precision' input
      statPresetInt { ExternalWritable := 'False'} : DInt;   //  Static value for the integer part of 'setup.preset' input
      statPresetDec { ExternalWritable := 'False'} : DInt;   //  Static value for the decimal part of 'setup.preset' input
   END_VAR

   VAR_TEMP 
      tempPulse : Bool;   //  Temporary value for 'pulse' input
      i : SInt;   //  Loop operand
   END_VAR

   VAR CONSTANT 
      ctSP_MAX_PRECISION : USInt := 6;   //  Constant value for maximum value of 'dt.precision'
   END_VAR


BEGIN
	REGION BLOCK HEADER
	    //===============================================================================
	    // CH / (c)Copyright (2023)
	    //-------------------------------------------------------------------------------
	    // Title:             (libMath_Total64REAL)
	    // Comment/Function:  (Big numbers capabilities with precision of max 6 decimals)
	    // Library/Family:    (Aktina\Tools\Math)
	    // Author:            (CH)
	    // Tested with:       (V16)
	    // Engineering:       (TIA Step7 Professional V16)
	    // Restrictions:      ()
	    // Requirements:      (S7 CPUs)
	    // Notes:             ()
	    //-------------------------------------------------------------------------------
	    // Change log table:
	    // Version  | Date       | Dev in charge          | Changes
	    //----------|------------|------------------------|------------------------------
	    // 01.00.00 | 2023-02-06 | (CH)                   | First released version
	    //===============================================================================
	END_REGION
	
	REGION BLOCK NOTES
	    //===============================================================================
	    
	    //===============================================================================
	END_REGION
	
	REGION GENERIC PRE-INSTRUCTIONS
	    // Work with temporary value / create process image
	    #tempPulse := #pulse;
	    
	    // Reset totalizer
	    IF (#dt.reset = TRUE) THEN
	        #dt.output := 0.0;
	    END_IF;
	    
	END_REGION GENERIC PRE-INSTRUCTIONS
	
	REGION REFRESH PRESET SETUP
	    // Calculate power of 10 (max = 8)
	    IF (#statPreset <> #dt.preset) OR (#statPrecision <> #dt.precision)
	        OR (#statTotal <> #dt.output)
	        OR (#refresh = TRUE) OR (#dt.reset = TRUE)
	    THEN
	        
	        IF #dt.precision > #ctSP_MAX_PRECISION THEN
	            #dt.precision := #ctSP_MAX_PRECISION;
	        END_IF;
	        
	        #statExp := LREAL_TO_DINT(10 ** #dt.precision);
	        
	        // Calculate preset addition based on precision
	        #statPresetInt := TRUNC_DINT(IN := #dt.preset);
	        #statPresetDec := TRUNC_DINT((#dt.preset - DINT_TO_REAL(#statPresetInt)) * DINT_TO_REAL(#statExp));
	        
	        #statTotal := #dt.output;
	        
	        #statTotalInt := TRUNC_DINT(IN := #statTotal);
	        #statTotalDec := TRUNC_DINT((#statTotal - DINT_TO_LREAL(#statTotalInt)) * DINT_TO_LREAL(#statExp));
	        
	        #statPreset := #dt.preset;
	        #statPrecision := #dt.precision;
	        
	        #statValid := #statPresetDec < #statExp;
	        
	    END_IF;
	    
	END_REGION REFRESH PRESET SETUP
	
	REGION TOTALIZER
	    
	    IF (#tempPulse = TRUE) AND (#statPulseOld = FALSE) // edge only
	        AND (#dt.preset > 0)
	        AND (#dt.reset = FALSE) // when force jobs are enabled we by-pass the totalizer
	        AND (#statValid = TRUE)
	    THEN
	        
	        #statTotalDec := #statTotalDec + #statPresetDec;
	        IF #statTotalDec >= #statExp THEN
	            #statTotalInt := #statTotalInt + 1;
	            #statTotalDec := #statTotalDec - #statExp;
	            
	        END_IF;
	        
	        #statTotalInt := #statTotalInt + #statPresetInt;
	        
	    END_IF;
	    
	    // Edge logic
	    #statPulseOld := #tempPulse;
	    
	END_REGION TOTALIZER
	
	REGION OUTPUTS
	    // Synth total value
	    #statTotal := DINT_TO_LREAL(#statTotalInt) + (DINT_TO_LREAL(#statTotalDec) / #statExp);
	    
	    // Write static value to output
	    #dt.output := #statTotal;
	    
	END_REGION OUTPUTS
END_FUNCTION_BLOCK

FUNCTION_BLOCK "AFB_OptionCtrl"
TITLE = AFB_OptionCtrl
{ S7_Optimized_Access := 'TRUE' }
AUTHOR : CH
FAMILY : Aktina
NAME : Operator
VERSION : 0.1
//AFB_OptionCtrl
   VAR_INPUT 
      number : Int;   //  Number of options to scan (cannot exceed CT_MAX_OPTIONS)
      optIn : Array[0..#ctARRAY_OPTION] of "typeOptionIn";   //  Array of all options incoming conditions from sequencers and environment
   END_VAR

   VAR_OUTPUT 
      availAct3Mains : Bool;   //  TRUE: Provide an action 1 - 4 (start - stop - end, all highight dependent)
      availActCancel : Bool;   //  TRUE: Provide an action 8 (cancel all)
      availActConfirm : Bool;   //  TRUE: Provide an action 16 (confirm, highight dependent)
      availActResetTime : Bool;   //  TRUE: Provide an action 32 (reset time, highlight dependent)
   END_VAR

   VAR_IN_OUT 
      action : Int;   //  Actions from the operation center (0-none, 1=start, 2=stop, 4=end, 8=cancel, 16=confirm)
      optOut : Array[0..#ctARRAY_OPTION] of "typeOptionOut";   //  Array of all options outgoing conditions & status
   END_VAR

   VAR 
      statNumber : Int;   //  Static value for the "number" input
      statDetChange : Array[0..#ctARRAY_OPTION] of Byte;   //  Static array of bytes used to detect changes in options status
      statAction : Struct   //  Temporary struct used to translate the action int to bits
         bit8 : Bool;
         bit9 : Bool;
         bit10 : Bool;
         bit11 : Bool;
         bit12 : Bool;
         bit13 : Bool;
         bit14 : Bool;
         bit15 : Bool;
         start : Bool;
         stop : Bool;
         end : Bool;
         cancel : Bool;
         confirm : Bool;
         resetTime : Bool;
         bit6 : Bool;
         bit7 : Bool;
      END_STRUCT;
      statAvailAct3Mains : Bool;   //  Static bit for "availAct3Mains" output
      statAvailActCancel : Bool;   //  Static bit for "availActCancel" output
      statAvailActConfirm : Bool;   //  Static bit for "availActConfirm" output
      statAvailActResetTime : Bool;   //  Static bit for "availActResetTime" output
      bufferTOFs {InstructionName := 'IEC_TIMER'; LibVersion := '1.0'; S7_SetPoint := 'False'} : Array[0..#ctARRAY_OPTION] of IEC_TIMER;   //  Static group of highlight timers buffers
      instTimer {InstructionName := 'IEC_TIMER'; LibVersion := '1.0'; ExternalAccessible := 'False'; ExternalVisible := 'False'; ExternalWritable := 'False'; S7_SetPoint := 'False'} : IEC_TIMER;   //  Instance timer used for all highlights
   END_VAR

   VAR_TEMP 
      tempN : Int;   //  Temporary "n" loop operand
      tempIn : "typeOptionIn";   //  Temporary memory area for the "optBitsIn" input (read only)
      tempOut : "typeOptionOut";   //  Temporary memory area for the "optBitsOut" output (read & write)
      tempStatus : Word;   //  Temporary status buffer
      tempAction : Word;   //  Temporary memory area for the "action" inout
      tempDetectBefore : Byte;   //  Temporary status change detection buffer before program execution (used to reset highlights individually)
      tempDetectAfter : Byte;   //  Temporary status change detection buffer after program execution (used to reset highlights individually)
      tempDetAllow1to4 : Bool;   //  Temporary bit used to detect an active highlight to allow actions 1 to 4
      tempDetAllow8 : Bool;   //  Temporary bit used to detect an active procedure to allow action 8
      tempDetAllow16 : Bool;   //  Temporary bit used to detect an active highlight and prompt to allow action 16
      tempDetAllow32 : Bool;   //  Temporary bit used to detect an active highlight and timeout to allow action 32
   END_VAR

   VAR CONSTANT 
      ctARRAY_OPTION : Int := 7;   //  Constant value for the arrays upper limit (CT_MAX_OPTIONS - 1)
      ctMAX_OPTIONS : Int := 8;   //  Constant value for the maximum option number (better handle as 8, 16, 32 etc)
      ctNULL : Word := 16#0000;   //  Constant Word = 16#0
   END_VAR


BEGIN
	REGION BLOCK HEADER
	    //===============================================================================
	    // CH / (c)Copyright (2021)
	    //-------------------------------------------------------------------------------
	    // Title:             (Options Control)
	    // Comment/Function:  (Control multiple options using the same set of action keys)
	    // Library/Family:    (Aktina/Tools/Operation)
	    // Author:            (CH)
	    // Tested with:       (V16)
	    // Engineering:       (TIA Step7 Professional V16)
	    // Restrictions:      ()
	    // Requirements:      (S7-15xx/12xx CPUs)
	    // Notes:             (See block notes)
	    //-------------------------------------------------------------------------------
	    // Change log table:
	    // Version  | Date       | Dev in charge          | Changes
	    //----------|------------|------------------------|------------------------------
	    // 01.00.00 | 2021-07-27 | (CH)                   | First released version
	    //===============================================================================
	END_REGION
	
	REGION BLOCK NOTES
	    //===============================================================================
	    // 1: The number of options participating is configured by the CT_MAX_OPTION
	    //-------------------------------------------------------------------------------
	    // 2: Each option has a group of status bits and a unique status number that
	    // transfer the information to the operation center
	    //===============================================================================
	END_REGION
	
	REGION GENERIC PRE-INSTRUCTIONS
	    // Init temporary area
	    #tempN := 0;
	    "AFC_Word_To_Struct"(w := #ctNULL,
	                         s => #tempIn.cond);
	    #tempIn.tof := 0;
	    #tempOut.cond := #tempIn.cond;
	    #tempOut.status := 0;
	    #tempStatus := 0;
	    #tempDetectBefore := 0;
	    #tempDetectAfter := 0;
	    #tempDetAllow1to4 := FALSE;
	    #tempDetAllow8 := FALSE;
	    
	    // Import and evaluate number of options
	    IF (#number <= #ctMAX_OPTIONS) AND (#number >= 0)
	    THEN // write input to stat unchanged
	        #statNumber := #number;
	    ELSIF (#number > #ctMAX_OPTIONS)
	    THEN // automatically adapt maximum options number to the static variable
	        #statNumber := #ctMAX_OPTIONS;
	    ELSE // in any other case write 0 to stat
	        #statNumber := 0;
	    END_IF;
	    
	    // Transfer actions int to bit
	    "AFC_Word_To_Struct"(w := INT_TO_WORD(#action),
	                         s => #statAction);
	    
	END_REGION GENERIC PRE-INSTRUCTIONS
	
	REGION CONTROL OPTIONS
	    
	    IF #statNumber > 0
	    THEN // Run the loop only if there is a reason. If there are no options then stop it
	        
	        FOR #tempN := 0 TO (#statNumber - 1) DO
	            
	            REGION import data to scanned instance
	                // Import: Saved data to temporary memory area
	                #tempDetectBefore := #statDetChange[#tempN];
	                
	                #tempIn := #optIn[#tempN];
	                #tempOut := #optOut[#tempN];
	                
	                // Load timer
	                PRESET_TIMER(PT := DINT_TO_TIME(#tempIn.tof),
	                             TIMER := #bufferTOFs[#tempN]);
	                
	                #instTimer := #bufferTOFs[#tempN];
	                
	            END_REGION import data to scanned instance
	            
	            REGION create output conditions
	                // Status: Option relevant error
	                #tempOut.cond.error := (#tempIn.cond.ongoing = TRUE) AND (#tempIn.cond.error = TRUE);
	                
	                // Status: Block option from starting
	                #tempOut.cond.block := (#tempIn.cond.block = TRUE); // AND (#tempIn.cond.ongoing = FALSE)
	                
	                // Timer: Highlight
	                #instTimer.TOF(IN := (#tempIn.cond.highlight = TRUE)
	                               AND (((#tempOut.cond.block = FALSE) AND (#tempIn.cond.error = FALSE))
	                               OR ((#tempIn.cond.ongoing = TRUE) AND (#tempOut.cond.endCond = FALSE))),
	                               PT := #instTimer.PT);
	                
	                // Status: Highlight
	                #tempOut.cond.highlight := #instTimer.Q;
	                
	                // Status: Start condition (hold till highlight is reset or process is set)
	                #tempOut.cond.startCond := (((#tempOut.cond.highlight = TRUE) AND ((#statAction.start = TRUE) OR (#tempOut.cond.startCond = TRUE)))
	                OR (#tempIn.cond.extStart = TRUE))
	                AND (#tempIn.cond.ongoing = FALSE)
	                AND NOT ((#tempOut.cond.highlight = TRUE) AND ((#statAction.stop = TRUE) OR (#statAction.end = TRUE)))
	                AND NOT (#statAction.cancel = TRUE) AND NOT (#tempIn.cond.extCancel = TRUE)
	                ;
	                
	                // Status: Run (hold till error, end or pause)
	                #tempOut.cond.run := (#tempIn.cond.ongoing = TRUE) AND (#tempIn.cond.error = FALSE)
	                AND NOT ((#tempOut.cond.highlight = TRUE) AND ((#statAction.stop = TRUE) OR (#statAction.end = TRUE))) AND NOT (#statAction.cancel = TRUE)
	                AND ((#tempOut.cond.run = TRUE) OR ((#tempOut.cond.highlight = TRUE) AND (#statAction.start = TRUE)) OR (#tempIn.cond.extStart = TRUE));
	                
	                // Status: Hibernate (invert run)
	                #tempOut.cond.hibernate := (#tempIn.cond.ongoing = TRUE) AND (#tempOut.cond.run = FALSE);
	                
	                // Status: End condition
	                #tempOut.cond.endCond := (#tempIn.cond.ongoing = TRUE)
	                AND (((#tempOut.cond.highlight = TRUE) AND (#statAction.end = TRUE)) OR (#statAction.cancel = TRUE) OR (#tempOut.cond.endCond = TRUE));
	                
	                // Status: Timed out
	                #tempOut.cond.timeout := (#tempIn.cond.ongoing = TRUE) AND (#tempIn.cond.timeout = TRUE);
	                
	                // Status: Prompt for confirmation
	                #tempOut.cond.prompt := (#tempIn.cond.ongoing = TRUE) AND (#tempIn.cond.prompt = TRUE);
	                
	                // Status: Confirmation acknowledgement
	                #tempOut.cond.confirm := (#tempIn.cond.ongoing = TRUE) AND (#tempOut.cond.prompt = TRUE) AND (#statAction.confirm = TRUE);
	                
	                // Status: Timeout acknowledgement
	                #tempOut.cond.resetTime := (#tempIn.cond.ongoing = TRUE) AND (#tempOut.cond.timeout = TRUE) AND (#tempOut.cond.highlight = TRUE) AND (#statAction.resetTime = TRUE);
	                
	                // Status: Collective integer
	                "AFC_Struct_To_Word"(s := #tempOut.cond,
	                                     w => #tempStatus);
	                
	                #tempOut.status := WORD_TO_UINT(#tempStatus);
	                
	            END_REGION create output conditions
	            
	            REGION actions allowance
	                // Detect: Change in run or enabled (used to reset highlight)
	                #tempDetectAfter := 16#0;
	                #tempDetectAfter.%X0 := #tempIn.cond.ongoing;
	                #tempDetectAfter.%X1 := #tempOut.cond.run;
	                #tempDetectAfter.%X2 := #tempOut.cond.prompt;
	                
	                IF (#tempDetectBefore <> #tempDetectAfter) OR (#tempOut.cond.block = TRUE) OR (#tempOut.cond.highlight = TRUE AND (#statAction.end = TRUE)) OR (#statAction.cancel = TRUE)
	                THEN
	                    RESET_TIMER(#instTimer);
	                    #tempOut.cond.highlight := false;
	                END_IF;
	                
	                // Detect: Allow commands 1 to 4
	                IF (#tempOut.cond.highlight = TRUE)
	                THEN
	                    #tempDetAllow1to4 := TRUE;
	                END_IF;
	                
	                // Detect: Allow command 8
	                IF (#tempIn.cond.ongoing = TRUE) OR (#tempOut.cond.highlight = TRUE)
	                THEN
	                    #tempDetAllow8 := TRUE;
	                END_IF;
	                
	                // Detect: Allow command 16
	                IF (#tempOut.cond.prompt = TRUE)
	                THEN
	                    #tempDetAllow16 := TRUE;
	                END_IF;
	                
	                // Detect: Allow command 32
	                IF (#tempOut.cond.timeout = TRUE)
	                THEN
	                    #tempDetAllow32 := TRUE;
	                END_IF;
	                
	            END_REGION actions allowance
	            
	            REGION export data to scanned instance
	                // Return: Save data
	                #optOut[#tempN] := #tempOut;
	                #bufferTOFs[#tempN] := #instTimer;
	                #statDetChange[#tempN] := #tempDetectAfter;
	                
	            END_REGION export data TO scanned INSTANCE  
	            
	        END_FOR;
	        
	    END_IF;
	    
	    REGION reset inactive options data
	        // Run the loop to reset the remaining not used options
	        FOR #tempN := #statNumber TO #ctARRAY_OPTION DO
	            
	            "AFC_Word_To_Struct"(w := #ctNULL,
	                                 s => #tempOut.cond);
	            
	            #tempStatus := 16#0;
	            #tempOut.status := WORD_TO_UINT(#tempStatus);
	            
	            // Return temporary data to runtime data
	            #optOut[#tempN] := #tempOut;
	            
	            RESET_TIMER(#bufferTOFs[#tempN]);
	            
	        END_FOR;
	        
	    END_REGION reset inactive "Options" data
	    
	    REGION reset availability and latching buttons
	        // Static: Allow commands
	        #statAvailAct3Mains := (#tempDetAllow1to4 = TRUE);
	        #statAvailActCancel := (#tempDetAllow8 = TRUE);
	        #statAvailActConfirm := (#tempDetAllow16 = TRUE);
	        #statAvailActResetTime := (#tempDetAllow32 = TRUE);
	        
